    RBT4_STANDARD_WELD_DATA : WORD ;
    RBT5_STANDARD_WELD_DATA : WORD ;
    RBT6_STANDARD_WELD_DATA : WORD ;
    RBT7_STANDARD_WELD_DATA : WORD ;
    RBT8_STANDARD_WELD_DATA : WORD ;
    RBT9_STANDARD_WELD_DATA : WORD ;
    RBT10_STANDARD_WELD_DATA : WORD ;
    RBT11_STANDARD_WELD_DATA : WORD ;
    RBT12_STANDARD_WELD_DATA : WORD ;
    RBT13_STANDARD_WELD_DATA : WORD ;
    RBT14_STANDARD_WELD_DATA : WORD ;
    RBT15_STANDARD_WELD_DATA : WORD ;
    RBT16_STANDARD_WELD_DATA : WORD ;
    RBT17_STANDARD_WELD_DATA : WORD ;
    RBT18_STANDARD_WELD_DATA : WORD ;
    RBT19_STANDARD_WELD_DATA : WORD ;
    RBT20_STANDARD_WELD_DATA : WORD ;
    RBT21_STANDARD_WELD_DATA : WORD ;
    RBT22_STANDARD_WELD_DATA : WORD ;
    RBT23_STANDARD_WELD_DAT : WORD ;
    RBT24_STANDARD_WELD_DAT : WORD ;
    CHK_WORD : WORD ;
    TEST_TEMP : ARRAY  [1 .. 40 ] OF BYTE ;
   END_STRUCT ;
   S701_BT_CODE_2016 : STRUCT
    STATION_MAIN : WORD ;
    DISTINCTION_LH_RH : WORD ;
    STAION_NUMBER : WORD ;
    BODY_TYPE_1ST : WORD ;
    BODY_TYPE_OPTION : WORD ;
    RBT1_STANDARD_WELD_DATA : WORD ;
    RBT2_STANDARD_WELD_DATA : WORD ;
    RBT3_STANDARD_WELD_DATA : WORD ;
    RBT4_STANDARD_WELD_DATA : WORD ;
    RBT5_STANDARD_WELD_DATA : WORD ;
    RBT6_STANDARD_WELD_DATA : WORD ;
    RBT7_STANDARD_WELD_DATA : WORD ;
    RBT8_STANDARD_WELD_DATA : WORD ;
    RBT9_STANDARD_WELD_DATA : WORD ;
    RBT10_STANDARD_WELD_DATA : WORD ;
    RBT11_STANDARD_WELD_DATA : WORD ;
    RBT12_STANDARD_WELD_DATA : WORD ;
    RBT13_STANDARD_WELD_DATA : WORD ;
    RBT14_STANDARD_WELD_DATA : WORD ;
    RBT15_STANDARD_WELD_DATA : WORD ;
    RBT16_STANDARD_WELD_DATA : WORD ;
    RBT17_STANDARD_WELD_DATA : WORD ;
    RBT18_STANDARD_WELD_DATA : WORD ;
    RBT19_STANDARD_WELD_DATA : WORD ;
    RBT20_STANDARD_WELD_DATA : WORD ;
    RBT21_STANDARD_WELD_DATA : WORD ;
    RBT22_STANDARD_WELD_DATA : WORD ;
    RBT23_STANDARD_WELD_DAT : WORD ;
    RBT24_STANDARD_WELD_DAT : WORD ;
    CHK_WORD : WORD ;
    TEST_TEMP : ARRAY  [1 .. 40 ] OF BYTE ;
   END_STRUCT ;
   S701_BT_CODE_2017 : STRUCT
    STATION_MAIN : WORD ;
    DISTINCTION_LH_RH : WORD ;
    STAION_NUMBER : WORD ;
    BODY_TYPE_1ST : WORD ;
    BODY_TYPE_OPTION : WORD ;
    RBT1_STANDARD_WELD_DATA : WORD ;
    RBT2_STANDARD_WELD_DATA : WORD ;
    RBT3_STANDARD_WELD_DATA : WORD ;
    RBT4_STANDARD_WELD_DATA : WORD ;
    RBT5_STANDARD_WELD_DATA : WORD ;
    RBT6_STANDARD_WELD_DATA : WORD ;
    RBT7_STANDARD_WELD_DATA : WORD ;
    RBT8_STANDARD_WELD_DATA : WORD ;
    RBT9_STANDARD_WELD_DATA : WORD ;
    RBT10_STANDARD_WELD_DATA : WORD ;
    RBT11_STANDARD_WELD_DATA : WORD ;
    RBT12_STANDARD_WELD_DATA : WORD ;
    RBT13_STANDARD_WELD_DATA : WORD ;
    RBT14_STANDARD_WELD_DATA : WORD ;
    RBT15_STANDARD_WELD_DATA : WORD ;
    RBT16_STANDARD_WELD_DATA : WORD ;
    RBT17_STANDARD_WELD_DATA : WORD ;
    RBT18_STANDARD_WELD_DATA : WORD ;
    RBT19_STANDARD_WELD_DATA : WORD ;
    RBT20_STANDARD_WELD_DATA : WORD ;
    RBT21_STANDARD_WELD_DATA : WORD ;
    RBT22_STANDARD_WELD_DATA : WORD ;
    RBT23_STANDARD_WELD_DAT : WORD ;
    RBT24_STANDARD_WELD_DAT : WORD ;
    CHK_WORD : WORD ;
    TEST_TEMP : ARRAY  [1 .. 40 ] OF BYTE ;
   END_STRUCT ;
   S701_BT_CODE_2018 : STRUCT
    STATION_MAIN : WORD ;
    DISTINCTION_LH_RH : WORD ;
    STAION_NUMBER : WORD ;
    BODY_TYPE_1ST : WORD ;
    BODY_TYPE_OPTION : WORD ;
    RBT1_STANDARD_WELD_DATA : WORD ;
    RBT2_STANDARD_WELD_DATA : WORD ;
    RBT3_STANDARD_WELD_DATA : WORD ;
    RBT4_STANDARD_WELD_DATA : WORD ;
    RBT5_STANDARD_WELD_DATA : WORD ;
    RBT6_STANDARD_WELD_DATA : WORD ;
    RBT7_STANDARD_WELD_DATA : WORD ;
    RBT8_STANDARD_WELD_DATA : WORD ;
    RBT9_STANDARD_WELD_DATA : WORD ;
    RBT10_STANDARD_WELD_DATA : WORD ;
    RBT11_STANDARD_WELD_DATA : WORD ;
    RBT12_STANDARD_WELD_DATA : WORD ;
    RBT13_STANDARD_WELD_DATA : WORD ;
    RBT14_STANDARD_WELD_DATA : WORD ;
    RBT15_STANDARD_WELD_DATA : WORD ;
    RBT16_STANDARD_WELD_DATA : WORD ;
    RBT17_STANDARD_WELD_DATA : WORD ;
    RBT18_STANDARD_WELD_DATA : WORD ;
    RBT19_STANDARD_WELD_DATA : WORD ;
    RBT20_STANDARD_WELD_DATA : WORD ;
    RBT21_STANDARD_WELD_DATA : WORD ;
    RBT22_STANDARD_WELD_DATA : WORD ;
    RBT23_STANDARD_WELD_DAT : WORD ;
    RBT24_STANDARD_WELD_DAT : WORD ;
    CHK_WORD : WORD ;
    TEST_TEMP : ARRAY  [1 .. 40 ] OF BYTE ;
   END_STRUCT ;
   S701_BT_CODE_2019 : STRUCT
    STATION_MAIN : WORD ;
    DISTINCTION_LH_RH : WORD ;
    STAION_NUMBER : WORD ;
    BODY_TYPE_1ST : WORD ;
    BODY_TYPE_OPTION : WORD ;
    RBT1_STANDARD_WELD_DATA : WORD ;
    RBT2_STANDARD_WELD_DATA : WORD ;
    RBT3_STANDARD_WELD_DATA : WORD ;
    RBT4_STANDARD_WELD_DATA : WORD ;
    RBT5_STANDARD_WELD_DATA : WORD ;
    RBT6_STANDARD_WELD_DATA : WORD ;
    RBT7_STANDARD_WELD_DATA : WORD ;
    RBT8_STANDARD_WELD_DATA : WORD ;
    RBT9_STANDARD_WELD_DATA : WORD ;
    RBT10_STANDARD_WELD_DATA : WORD ;
    RBT11_STANDARD_WELD_DATA : WORD ;
    RBT12_STANDARD_WELD_DATA : WORD ;
    RBT13_STANDARD_WELD_DATA : WORD ;
    RBT14_STANDARD_WELD_DATA : WORD ;
    RBT15_STANDARD_WELD_DATA : WORD ;
    RBT16_STANDARD_WELD_DATA : WORD ;
    RBT17_STANDARD_WELD_DATA : WORD ;
    RBT18_STANDARD_WELD_DATA : WORD ;
    RBT19_STANDARD_WELD_DATA : WORD ;
    RBT20_STANDARD_WELD_DATA : WORD ;
    RBT21_STANDARD_WELD_DATA : WORD ;
    RBT22_STANDARD_WELD_DATA : WORD ;
    RBT23_STANDARD_WELD_DAT : WORD ;
    RBT24_STANDARD_WELD_DAT : WORD ;
    CHK_WORD : WORD ;
    TEST_TEMP : ARRAY  [1 .. 40 ] OF BYTE ;
   END_STRUCT ;
   S701_BT_CODE_2020 : STRUCT
    STATION_MAIN : WORD ;
    DISTINCTION_LH_RH : WORD ;
    STAION_NUMBER : WORD ;
    BODY_TYPE_1ST : WORD ;
    BODY_TYPE_OPTION : WORD ;
    RBT1_STANDARD_WELD_DATA : WORD ;
    RBT2_STANDARD_WELD_DATA : WORD ;
    RBT3_STANDARD_WELD_DATA : WORD ;
    RBT4_STANDARD_WELD_DATA : WORD ;
    RBT5_STANDARD_WELD_DATA : WORD ;
    RBT6_STANDARD_WELD_DATA : WORD ;
    RBT7_STANDARD_WELD_DATA : WORD ;
    RBT8_STANDARD_WELD_DATA : WORD ;
    RBT9_STANDARD_WELD_DATA : WORD ;
    RBT10_STANDARD_WELD_DATA : WORD ;
    RBT11_STANDARD_WELD_DATA : WORD ;
    RBT12_STANDARD_WELD_DATA : WORD ;
    RBT13_STANDARD_WELD_DATA : WORD ;
    RBT14_STANDARD_WELD_DATA : WORD ;
    RBT15_STANDARD_WELD_DATA : WORD ;
    RBT16_STANDARD_WELD_DATA : WORD ;
    RBT17_STANDARD_WELD_DATA : WORD ;
    RBT18_STANDARD_WELD_DATA : WORD ;
    RBT19_STANDARD_WELD_DATA : WORD ;
    RBT20_STANDARD_WELD_DATA : WORD ;
    RBT21_STANDARD_WELD_DATA : WORD ;
    RBT22_STANDARD_WELD_DATA : WORD ;
    RBT23_STANDARD_WELD_DAT : WORD ;
    RBT24_STANDARD_WELD_DAT : WORD ;
    CHK_WORD : WORD ;
    TEST_TEMP : ARRAY  [1 .. 40 ] OF BYTE ;
   END_STRUCT ;
   S701_BT_CODE_2021 : STRUCT
    STATION_MAIN : WORD ;
    DISTINCTION_LH_RH : WORD ;
    STAION_NUMBER : WORD ;
    BODY_TYPE_1ST : WORD ;
    BODY_TYPE_OPTION : WORD ;
    RBT1_STANDARD_WELD_DATA : WORD ;
    RBT2_STANDARD_WELD_DATA : WORD ;
    RBT3_STANDARD_WELD_DATA : WORD ;
    RBT4_STANDARD_WELD_DATA : WORD ;
    RBT5_STANDARD_WELD_DATA : WORD ;
    RBT6_STANDARD_WELD_DATA : WORD ;
    RBT7_STANDARD_WELD_DATA : WORD ;
    RBT8_STANDARD_WELD_DATA : WORD ;
    RBT9_STANDARD_WELD_DATA : WORD ;
    RBT10_STANDARD_WELD_DATA : WORD ;
    RBT11_STANDARD_WELD_DATA : WORD ;
    RBT12_STANDARD_WELD_DATA : WORD ;
    RBT13_STANDARD_WELD_DATA : WORD ;
    RBT14_STANDARD_WELD_DATA : WORD ;
    RBT15_STANDARD_WELD_DATA : WORD ;
    RBT16_STANDARD_WELD_DATA : WORD ;
    RBT17_STANDARD_WELD_DATA : WORD ;
    RBT18_STANDARD_WELD_DATA : WORD ;
    RBT19_STANDARD_WELD_DATA : WORD ;
    RBT20_STANDARD_WELD_DATA : WORD ;
    RBT21_STANDARD_WELD_DATA : WORD ;
    RBT22_STANDARD_WELD_DATA : WORD ;
    RBT23_STANDARD_WELD_DAT : WORD ;
    RBT24_STANDARD_WELD_DAT : WORD ;
    CHK_WORD : WORD ;
    TEST_TEMP : ARRAY  [1 .. 40 ] OF BYTE ;
   END_STRUCT ;
   S701_BT_CODE_2022 : STRUCT
    STATION_MAIN : WORD ;
    DISTINCTION_LH_RH : WORD ;
    STAION_NUMBER : WORD ;
    BODY_TYPE_1ST : WORD ;
    BODY_TYPE_OPTION : WORD ;
    RBT1_STANDARD_WELD_DATA : WORD ;
    RBT2_STANDARD_WELD_DATA : WORD ;
    RBT3_STANDARD_WELD_DATA : WORD ;
    RBT4_STANDARD_WELD_DATA : WORD ;
    RBT5_STANDARD_WELD_DATA : WORD ;
    RBT6_STANDARD_WELD_DATA : WORD ;
    RBT7_STANDARD_WELD_DATA : WORD ;
    RBT8_STANDARD_WELD_DATA : WORD ;
    RBT9_STANDARD_WELD_DATA : WORD ;
    RBT10_STANDARD_WELD_DATA : WORD ;
    RBT11_STANDARD_WELD_DATA : WORD ;
    RBT12_STANDARD_WELD_DATA : WORD ;
    RBT13_STANDARD_WELD_DATA : WORD ;
    RBT14_STANDARD_WELD_DATA : WORD ;
    RBT15_STANDARD_WELD_DATA : WORD ;
    RBT16_STANDARD_WELD_DATA : WORD ;
    RBT17_STANDARD_WELD_DATA : WORD ;
    RBT18_STANDARD_WELD_DATA : WORD ;
    RBT19_STANDARD_WELD_DATA : WORD ;
    RBT20_STANDARD_WELD_DATA : WORD ;
    RBT21_STANDARD_WELD_DATA : WORD ;
    RBT22_STANDARD_WELD_DATA : WORD ;
    RBT23_STANDARD_WELD_DAT : WORD ;
    RBT24_STANDARD_WELD_DAT : WORD ;
    CHK_WORD : WORD ;
    TEST_TEMP : ARRAY  [1 .. 40 ] OF BYTE ;
   END_STRUCT ;
   S701_BT_CODE_2023 : STRUCT
    STATION_MAIN : WORD ;
    DISTINCTION_LH_RH : WORD ;
    STAION_NUMBER : WORD ;
    BODY_TYPE_1ST : WORD ;
    BODY_TYPE_OPTION : WORD ;
    RBT1_STANDARD_WELD_DATA : WORD ;
    RBT2_STANDARD_WELD_DATA : WORD ;
    RBT3_STANDARD_WELD_DATA : WORD ;
    RBT4_STANDARD_WELD_DATA : WORD ;
    RBT5_STANDARD_WELD_DATA : WORD ;
    RBT6_STANDARD_WELD_DATA : WORD ;
    RBT7_STANDARD_WELD_DATA : WORD ;
    RBT8_STANDARD_WELD_DATA : WORD ;
    RBT9_STANDARD_WELD_DATA : WORD ;
    RBT10_STANDARD_WELD_DATA : WORD ;
    RBT11_STANDARD_WELD_DATA : WORD ;
    RBT12_STANDARD_WELD_DATA : WORD ;
    RBT13_STANDARD_WELD_DATA : WORD ;
    RBT14_STANDARD_WELD_DATA : WORD ;
    RBT15_STANDARD_WELD_DATA : WORD ;
    RBT16_STANDARD_WELD_DATA : WORD ;
    RBT17_STANDARD_WELD_DATA : WORD ;
    RBT18_STANDARD_WELD_DATA : WORD ;
    RBT19_STANDARD_WELD_DATA : WORD ;
    RBT20_STANDARD_WELD_DATA : WORD ;
    RBT21_STANDARD_WELD_DATA : WORD ;
    RBT22_STANDARD_WELD_DATA : WORD ;
    RBT23_STANDARD_WELD_DAT : WORD ;
    RBT24_STANDARD_WELD_DAT : WORD ;
    CHK_WORD : WORD ;
    TEST_TEMP : ARRAY  [1 .. 40 ] OF BYTE ;
   END_STRUCT ;
   S701_BT_CODE_2024 : STRUCT
    STATION_MAIN : WORD ;
    DISTINCTION_LH_RH : WORD ;
    STAION_NUMBER : WORD ;
    BODY_TYPE_1ST : WORD ;
    BODY_TYPE_OPTION : WORD ;
    RBT1_STANDARD_WELD_DATA : WORD ;
    RBT2_STANDARD_WELD_DATA : WORD ;
    RBT3_STANDARD_WELD_DATA : WORD ;
    RBT4_STANDARD_WELD_DATA : WORD ;
    RBT5_STANDARD_WELD_DATA : WORD ;
    RBT6_STANDARD_WELD_DATA : WORD ;
    RBT7_STANDARD_WELD_DATA : WORD ;
    RBT8_STANDARD_WELD_DATA : WORD ;
    RBT9_STANDARD_WELD_DATA : WORD ;
    RBT10_STANDARD_WELD_DATA : WORD ;
    RBT11_STANDARD_WELD_DATA : WORD ;
    RBT12_STANDARD_WELD_DATA : WORD ;
    RBT13_STANDARD_WELD_DATA : WORD ;
    RBT14_STANDARD_WELD_DATA : WORD ;
    RBT15_STANDARD_WELD_DATA : WORD ;
    RBT16_STANDARD_WELD_DATA : WORD ;
    RBT17_STANDARD_WELD_DATA : WORD ;
    RBT18_STANDARD_WELD_DATA : WORD ;
    RBT19_STANDARD_WELD_DATA : WORD ;
    RBT20_STANDARD_WELD_DATA : WORD ;
    RBT21_STANDARD_WELD_DATA : WORD ;
    RBT22_STANDARD_WELD_DATA : WORD ;
    RBT23_STANDARD_WELD_DAT : WORD ;
    RBT24_STANDARD_WELD_DAT : WORD ;
    CHK_WORD : WORD ;
    TEST_TEMP : ARRAY  [1 .. 40 ] OF BYTE ;
   END_STRUCT ;
   S701_BT_CODE_2025 : STRUCT
    STATION_MAIN : WORD ;
    DISTINCTION_LH_RH : WORD ;
    STAION_NUMBER : WORD ;
    BODY_TYPE_1ST : WORD ;
    BODY_TYPE_OPTION : WORD ;
    RBT1_STANDARD_WELD_DATA : WORD ;
    RBT2_STANDARD_WELD_DATA : WORD ;
    RBT3_STANDARD_WELD_DATA : WORD ;
    RBT4_STANDARD_WELD_DATA : WORD ;
    RBT5_STANDARD_WELD_DATA : WORD ;
    RBT6_STANDARD_WELD_DATA : WORD ;
    RBT7_STANDARD_WELD_DATA : WORD ;
    RBT8_STANDARD_WELD_DATA : WORD ;
    RBT9_STANDARD_WELD_DATA : WORD ;
    RBT10_STANDARD_WELD_DATA : WORD ;
    RBT11_STANDARD_WELD_DATA : WORD ;
    RBT12_STANDARD_WELD_DATA : WORD ;
    RBT13_STANDARD_WELD_DATA : WORD ;
    RBT14_STANDARD_WELD_DATA : WORD ;
    RBT15_STANDARD_WELD_DATA : WORD ;
    RBT16_STANDARD_WELD_DATA : WORD ;
    RBT17_STANDARD_WELD_DATA : WORD ;
    RBT18_STANDARD_WELD_DATA : WORD ;
    RBT19_STANDARD_WELD_DATA : WORD ;
    RBT20_STANDARD_WELD_DATA : WORD ;
    RBT21_STANDARD_WELD_DATA : WORD ;
    RBT22_STANDARD_WELD_DATA : WORD ;
    RBT23_STANDARD_WELD_DAT : WORD ;
    RBT24_STANDARD_WELD_DAT : WORD ;
    CHK_WORD : WORD ;
    TEST_TEMP : ARRAY  [1 .. 40 ] OF BYTE ;
   END_STRUCT ;
   S701_BT_CODE_2026 : STRUCT
    STATION_MAIN : WORD ;
    DISTINCTION_LH_RH : WORD ;
    STAION_NUMBER : WORD ;
    BODY_TYPE_1ST : WORD ;
    BODY_TYPE_OPTION : WORD ;
    RBT1_STANDARD_WELD_DATA : WORD ;
    RBT2_STANDARD_WELD_DATA : WORD ;
    RBT3_STANDARD_WELD_DATA : WORD ;
    RBT4_STANDARD_WELD_DATA : WORD ;
    RBT5_STANDARD_WELD_DATA : WORD ;
    RBT6_STANDARD_WELD_DATA : WORD ;
    RBT7_STANDARD_WELD_DATA : WORD ;
    RBT8_STANDARD_WELD_DATA : WORD ;
    RBT9_STANDARD_WELD_DATA : WORD ;
    RBT10_STANDARD_WELD_DATA : WORD ;
    RBT11_STANDARD_WELD_DATA : WORD ;
    RBT12_STANDARD_WELD_DATA : WORD ;
    RBT13_STANDARD_WELD_DATA : WORD ;
    RBT14_STANDARD_WELD_DATA : WORD ;
    RBT15_STANDARD_WELD_DATA : WORD ;
    RBT16_STANDARD_WELD_DATA : WORD ;
    RBT17_STANDARD_WELD_DATA : WORD ;
    RBT18_STANDARD_WELD_DATA : WORD ;
    RBT19_STANDARD_WELD_DATA : WORD ;
    RBT20_STANDARD_WELD_DATA : WORD ;
    RBT21_STANDARD_WELD_DATA : WORD ;
    RBT22_STANDARD_WELD_DATA : WORD ;
    RBT23_STANDARD_WELD_DAT : WORD ;
    RBT24_STANDARD_WELD_DAT : WORD ;
    CHK_WORD : WORD ;
    TEST_TEMP : ARRAY  [1 .. 40 ] OF BYTE ;
   END_STRUCT ;
   S701_BT_CODE_2027 : STRUCT
    STATION_MAIN : WORD ;
    DISTINCTION_LH_RH : WORD ;
    STAION_NUMBER : WORD ;
    BODY_TYPE_1ST : WORD ;
    BODY_TYPE_OPTION : WORD ;
    RBT1_STANDARD_WELD_DATA : WORD ;
    RBT2_STANDARD_WELD_DATA : WORD ;
    RBT3_STANDARD_WELD_DATA : WORD ;
    RBT4_STANDARD_WELD_DATA : WORD ;
    RBT5_STANDARD_WELD_DATA : WORD ;
    RBT6_STANDARD_WELD_DATA : WORD ;
    RBT7_STANDARD_WELD_DATA : WORD ;
    RBT8_STANDARD_WELD_DATA : WORD ;
    RBT9_STANDARD_WELD_DATA : WORD ;
    RBT10_STANDARD_WELD_DATA : WORD ;
    RBT11_STANDARD_WELD_DATA : WORD ;
    RBT12_STANDARD_WELD_DATA : WORD ;
    RBT13_STANDARD_WELD_DATA : WORD ;
    RBT14_STANDARD_WELD_DATA : WORD ;
    RBT15_STANDARD_WELD_DATA : WORD ;
    RBT16_STANDARD_WELD_DATA : WORD ;
    RBT17_STANDARD_WELD_DATA : WORD ;
    RBT18_STANDARD_WELD_DATA : WORD ;
    RBT19_STANDARD_WELD_DATA : WORD ;
    RBT20_STANDARD_WELD_DATA : WORD ;
    RBT21_STANDARD_WELD_DATA : WORD ;
    RBT22_STANDARD_WELD_DATA : WORD ;
    RBT23_STANDARD_WELD_DAT : WORD ;
    RBT24_STANDARD_WELD_DAT : WORD ;
    CHK_WORD : WORD ;
    TEST_TEMP : ARRAY  [1 .. 40 ] OF BYTE ;
   END_STRUCT ;
   S701_BT_CODE_2028 : STRUCT
    STATION_MAIN : WORD ;
    DISTINCTION_LH_RH : WORD ;
    STAION_NUMBER : WORD ;
    BODY_TYPE_1ST : WORD ;
    BODY_TYPE_OPTION : WORD ;
    RBT1_STANDARD_WELD_DATA : WORD ;
    RBT2_STANDARD_WELD_DATA : WORD ;
    RBT3_STANDARD_WELD_DATA : WORD ;
    RBT4_STANDARD_WELD_DATA : WORD ;
    RBT5_STANDARD_WELD_DATA : WORD ;
    RBT6_STANDARD_WELD_DATA : WORD ;
    RBT7_STANDARD_WELD_DATA : WORD ;
    RBT8_STANDARD_WELD_DATA : WORD ;
    RBT9_STANDARD_WELD_DATA : WORD ;
    RBT10_STANDARD_WELD_DATA : WORD ;
    RBT11_STANDARD_WELD_DATA : WORD ;
    RBT12_STANDARD_WELD_DATA : WORD ;
    RBT13_STANDARD_WELD_DATA : WORD ;
    RBT14_STANDARD_WELD_DATA : WORD ;
    RBT15_STANDARD_WELD_DATA : WORD ;
    RBT16_STANDARD_WELD_DATA : WORD ;
    RBT17_STANDARD_WELD_DATA : WORD ;
    RBT18_STANDARD_WELD_DATA : WORD ;
    RBT19_STANDARD_WELD_DATA : WORD ;
    RBT20_STANDARD_WELD_DATA : WORD ;
    RBT21_STANDARD_WELD_DATA : WORD ;
    RBT22_STANDARD_WELD_DATA : WORD ;
    RBT23_STANDARD_WELD_DAT : WORD ;
    RBT24_STANDARD_WELD_DAT : WORD ;
    CHK_WORD : WORD ;
    TEST_TEMP : ARRAY  [1 .. 40 ] OF BYTE ;
   END_STRUCT ;
   S701_BT_CODE_2029 : STRUCT
    STATION_MAIN : WORD ;
    DISTINCTION_LH_RH : WORD ;
    STAION_NUMBER : WORD ;
    BODY_TYPE_1ST : WORD ;
    BODY_TYPE_OPTION : WORD ;
    RBT1_STANDARD_WELD_DATA : WORD ;
    RBT2_STANDARD_WELD_DATA : WORD ;
    RBT3_STANDARD_WELD_DATA : WORD ;
    RBT4_STANDARD_WELD_DATA : WORD ;
    RBT5_STANDARD_WELD_DATA : WORD ;
    RBT6_STANDARD_WELD_DATA : WORD ;
    RBT7_STANDARD_WELD_DATA : WORD ;
    RBT8_STANDARD_WELD_DATA : WORD ;
    RBT9_STANDARD_WELD_DATA : WORD ;
    RBT10_STANDARD_WELD_DATA : WORD ;
    RBT11_STANDARD_WELD_DATA : WORD ;
    RBT12_STANDARD_WELD_DATA : WORD ;
    RBT13_STANDARD_WELD_DATA : WORD ;
    RBT14_STANDARD_WELD_DATA : WORD ;
    RBT15_STANDARD_WELD_DATA : WORD ;
    RBT16_STANDARD_WELD_DATA : WORD ;
    RBT17_STANDARD_WELD_DATA : WORD ;
    RBT18_STANDARD_WELD_DATA : WORD ;
    RBT19_STANDARD_WELD_DATA : WORD ;
    RBT20_STANDARD_WELD_DATA : WORD ;
    RBT21_STANDARD_WELD_DATA : WORD ;
    RBT22_STANDARD_WELD_DATA : WORD ;
    RBT23_STANDARD_WELD_DAT : WORD ;
    RBT24_STANDARD_WELD_DAT : WORD ;
    CHK_WORD : WORD ;
    TEST_TEMP : ARRAY  [1 .. 40 ] OF BYTE ;
   END_STRUCT ;
   S701_BT_CODE_2030 : STRUCT
    STATION_MAIN : WORD ;
    DISTINCTION_LH_RH : WORD ;
    STAION_NUMBER : WORD ;
    BODY_TYPE_1ST : WORD ;
    BODY_TYPE_OPTION : WORD ;
    RBT1_STANDARD_WELD_DATA : WORD ;
    RBT2_STANDARD_WELD_DATA : WORD ;
    RBT3_STANDARD_WELD_DATA : WORD ;
    RBT4_STANDARD_WELD_DATA : WORD ;
    RBT5_STANDARD_WELD_DATA : WORD ;
    RBT6_STANDARD_WELD_DATA : WORD ;
    RBT7_STANDARD_WELD_DATA : WORD ;
    RBT8_STANDARD_WELD_DATA : WORD ;
    RBT9_STANDARD_WELD_DATA : WORD ;
    RBT10_STANDARD_WELD_DATA : WORD ;
    RBT11_STANDARD_WELD_DATA : WORD ;
    RBT12_STANDARD_WELD_DATA : WORD ;
    RBT13_STANDARD_WELD_DATA : WORD ;
    RBT14_STANDARD_WELD_DATA : WORD ;
    RBT15_STANDARD_WELD_DATA : WORD ;
    RBT16_STANDARD_WELD_DATA : WORD ;
    RBT17_STANDARD_WELD_DATA : WORD ;
    RBT18_STANDARD_WELD_DATA : WORD ;
    RBT19_STANDARD_WELD_DATA : WORD ;
    RBT20_STANDARD_WELD_DATA : WORD ;
    RBT21_STANDARD_WELD_DATA : WORD ;
    RBT22_STANDARD_WELD_DATA : WORD ;
    RBT23_STANDARD_WELD_DAT : WORD ;
    RBT24_STANDARD_WELD_DAT : WORD ;
    CHK_WORD : WORD ;
    TEST_TEMP : ARRAY  [1 .. 40 ] OF BYTE ;
   END_STRUCT ;
   S700_BT_CODE_2101 : STRUCT
    STATION_MAIN : WORD ;
    DISTINCTION_LH_RH : WORD ;
    STAION_NUMBER : WORD ;
    BODY_TYPE_1ST : WORD ;
    BODY_TYPE_OPTION : WORD ;
    RBT1_STANDARD_WELD_DATA : WORD ;
    RBT2_STANDARD_WELD_DATA : WORD ;
    RBT3_STANDARD_WELD_DATA : WORD ;
    RBT4_STANDARD_WELD_DATA : WORD ;
    RBT5_STANDARD_WELD_DATA : WORD ;
    RBT6_STANDARD_WELD_DATA : WORD ;
    RBT7_STANDARD_WELD_DATA : WORD ;
    RBT8_STANDARD_WELD_DATA : WORD ;
    RBT9_STANDARD_WELD_DATA : WORD ;
    RBT10_STANDARD_WELD_DATA : WORD ;
    RBT11_STANDARD_WELD_DATA : WORD ;
    RBT12_STANDARD_WELD_DATA : WORD ;
    RBT13_STANDARD_WELD_DATA : WORD ;
    RBT14_STANDARD_WELD_DATA : WORD ;
    RBT15_STANDARD_WELD_DATA : WORD ;
    RBT16_STANDARD_WELD_DATA : WORD ;
    RBT17_STANDARD_WELD_DATA : WORD ;
    RBT18_STANDARD_WELD_DATA : WORD ;
    RBT19_STANDARD_WELD_DATA : WORD ;
    RBT20_STANDARD_WELD_DATA : WORD ;
    RBT21_STANDARD_WELD_DATA : WORD ;
    RBT22_STANDARD_WELD_DATA : WORD ;
    RBT23_STANDARD_WELD_DAT : WORD ;
    RBT24_STANDARD_WELD_DAT : WORD ;
    CHK_WORD : WORD ;
    TEST_TEMP : ARRAY  [1 .. 40 ] OF BYTE ;
   END_STRUCT ;
   S700_BT_CODE_2102 : STRUCT
    STATION_MAIN : WORD ;
    DISTINCTION_LH_RH : WORD ;
    STAION_NUMBER : WORD ;
    BODY_TYPE_1ST : WORD ;
    BODY_TYPE_OPTION : WORD ;
    RBT1_STANDARD_WELD_DATA : WORD ;
    RBT2_STANDARD_WELD_DATA : WORD ;
    RBT3_STANDARD_WELD_DATA : WORD ;
    RBT4_STANDARD_WELD_DATA : WORD ;
    RBT5_STANDARD_WELD_DATA : WORD ;
    RBT6_STANDARD_WELD_DATA : WORD ;
    RBT7_STANDARD_WELD_DATA : WORD ;
    RBT8_STANDARD_WELD_DATA : WORD ;
    RBT9_STANDARD_WELD_DATA : WORD ;
    RBT10_STANDARD_WELD_DATA : WORD ;
    RBT11_STANDARD_WELD_DATA : WORD ;
    RBT12_STANDARD_WELD_DATA : WORD ;
    RBT13_STANDARD_WELD_DATA : WORD ;
    RBT14_STANDARD_WELD_DATA : WORD ;
    RBT15_STANDARD_WELD_DATA : WORD ;
    RBT16_STANDARD_WELD_DATA : WORD ;
    RBT17_STANDARD_WELD_DATA : WORD ;
    RBT18_STANDARD_WELD_DATA : WORD ;
    RBT19_STANDARD_WELD_DATA : WORD ;
    RBT20_STANDARD_WELD_DATA : WORD ;
    RBT21_STANDARD_WELD_DATA : WORD ;
    RBT22_STANDARD_WELD_DATA : WORD ;
    RBT23_STANDARD_WELD_DAT : WORD ;
    RBT24_STANDARD_WELD_DAT : WORD ;
    CHK_WORD : WORD ;
    TEST_TEMP : ARRAY  [1 .. 40 ] OF BYTE ;
   END_STRUCT ;
   S700_BT_CODE_2103 : STRUCT
    STATION_MAIN : WORD ;
    DISTINCTION_LH_RH : WORD ;
    STAION_NUMBER : WORD ;
    BODY_TYPE_1ST : WORD ;
    BODY_TYPE_OPTION : WORD ;
    RBT1_STANDARD_WELD_DATA : WORD ;
    RBT2_STANDARD_WELD_DATA : WORD ;
    RBT3_STANDARD_WELD_DATA : WORD ;
    RBT4_STANDARD_WELD_DATA : WORD ;
    RBT5_STANDARD_WELD_DATA : WORD ;
    RBT6_STANDARD_WELD_DATA : WORD ;
    RBT7_STANDARD_WELD_DATA : WORD ;
    RBT8_STANDARD_WELD_DATA : WORD ;
    RBT9_STANDARD_WELD_DATA : WORD ;
    RBT10_STANDARD_WELD_DATA : WORD ;
    RBT11_STANDARD_WELD_DATA : WORD ;
    RBT12_STANDARD_WELD_DATA : WORD ;
    RBT13_STANDARD_WELD_DATA : WORD ;
    RBT14_STANDARD_WELD_DATA : WORD ;
    RBT15_STANDARD_WELD_DATA : WORD ;
    RBT16_STANDARD_WELD_DATA : WORD ;
    RBT17_STANDARD_WELD_DATA : WORD ;
    RBT18_STANDARD_WELD_DATA : WORD ;
    RBT19_STANDARD_WELD_DATA : WORD ;
    RBT20_STANDARD_WELD_DATA : WORD ;
    RBT21_STANDARD_WELD_DATA : WORD ;
    RBT22_STANDARD_WELD_DATA : WORD ;
    RBT23_STANDARD_WELD_DAT : WORD ;
    RBT24_STANDARD_WELD_DAT : WORD ;
    CHK_WORD : WORD ;
    TEST_TEMP : ARRAY  [1 .. 40 ] OF BYTE ;
   END_STRUCT ;
   S700_BT_CODE_2104 : STRUCT
    STATION_MAIN : WORD ;
    DISTINCTION_LH_RH : WORD ;
    STAION_NUMBER : WORD ;
    BODY_TYPE_1ST : WORD ;
    BODY_TYPE_OPTION : WORD ;
    RBT1_STANDARD_WELD_DATA : WORD ;
    RBT2_STANDARD_WELD_DATA : WORD ;
    RBT3_STANDARD_WELD_DATA : WORD ;
    RBT4_STANDARD_WELD_DATA : WORD ;
    RBT5_STANDARD_WELD_DATA : WORD ;
    RBT6_STANDARD_WELD_DATA : WORD ;
    RBT7_STANDARD_WELD_DATA : WORD ;
    RBT8_STANDARD_WELD_DATA : WORD ;
    RBT9_STANDARD_WELD_DATA : WORD ;
    RBT10_STANDARD_WELD_DATA : WORD ;
    RBT11_STANDARD_WELD_DATA : WORD ;
    RBT12_STANDARD_WELD_DATA : WORD ;
    RBT13_STANDARD_WELD_DATA : WORD ;
    RBT14_STANDARD_WELD_DATA : WORD ;
    RBT15_STANDARD_WELD_DATA : WORD ;
    RBT16_STANDARD_WELD_DATA : WORD ;
    RBT17_STANDARD_WELD_DATA : WORD ;
    RBT18_STANDARD_WELD_DATA : WORD ;
    RBT19_STANDARD_WELD_DATA : WORD ;
    RBT20_STANDARD_WELD_DATA : WORD ;
    RBT21_STANDARD_WELD_DATA : WORD ;
    RBT22_STANDARD_WELD_DATA : WORD ;
    RBT23_STANDARD_WELD_DAT : WORD ;
    RBT24_STANDARD_WELD_DAT : WORD ;
    CHK_WORD : WORD ;
    TEST_TEMP : ARRAY  [1 .. 40 ] OF BYTE ;
   END_STRUCT ;
   S700_BT_CODE_2105 : STRUCT
    STATION_MAIN : WORD ;
    DISTINCTION_LH_RH : WORD ;
    STAION_NUMBER : WORD ;
    BODY_TYPE_1ST : WORD ;
    BODY_TYPE_OPTION : WORD ;
    RBT1_STANDARD_WELD_DATA : WORD ;
    RBT2_STANDARD_WELD_DATA : WORD ;
    RBT3_STANDARD_WELD_DATA : WORD ;
    RBT4_STANDARD_WELD_DATA : WORD ;
    RBT5_STANDARD_WELD_DATA : WORD ;
    RBT6_STANDARD_WELD_DATA : WORD ;
    RBT7_STANDARD_WELD_DATA : WORD ;
    RBT8_STANDARD_WELD_DATA : WORD ;
    RBT9_STANDARD_WELD_DATA : WORD ;
    RBT10_STANDARD_WELD_DATA : WORD ;
    RBT11_STANDARD_WELD_DATA : WORD ;
    RBT12_STANDARD_WELD_DATA : WORD ;
    RBT13_STANDARD_WELD_DATA : WORD ;
    RBT14_STANDARD_WELD_DATA : WORD ;
    RBT15_STANDARD_WELD_DATA : WORD ;
    RBT16_STANDARD_WELD_DATA : WORD ;
    RBT17_STANDARD_WELD_DATA : WORD ;
    RBT18_STANDARD_WELD_DATA : WORD ;
    RBT19_STANDARD_WELD_DATA : WORD ;
    RBT20_STANDARD_WELD_DATA : WORD ;
    RBT21_STANDARD_WELD_DATA : WORD ;
    RBT22_STANDARD_WELD_DATA : WORD ;
    RBT23_STANDARD_WELD_DAT : WORD ;
    RBT24_STANDARD_WELD_DAT : WORD ;
    CHK_WORD : WORD ;
    TEST_TEMP : ARRAY  [1 .. 40 ] OF BYTE ;
   END_STRUCT ;
   S700_BT_CODE_2106 : STRUCT
    STATION_MAIN : WORD ;
    DISTINCTION_LH_RH : WORD ;
    STAION_NUMBER : WORD ;
    BODY_TYPE_1ST : WORD ;
    BODY_TYPE_OPTION : WORD ;
    RBT1_STANDARD_WELD_DATA : WORD ;
    RBT2_STANDARD_WELD_DATA : WORD ;
    RBT3_STANDARD_WELD_DATA : WORD ;
    RBT4_STANDARD_WELD_DATA : WORD ;
    RBT5_STANDARD_WELD_DATA : WORD ;
    RBT6_STANDARD_WELD_DATA : WORD ;
    RBT7_STANDARD_WELD_DATA : WORD ;
    RBT8_STANDARD_WELD_DATA : WORD ;
    RBT9_STANDARD_WELD_DATA : WORD ;
    RBT10_STANDARD_WELD_DATA : WORD ;
    RBT11_STANDARD_WELD_DATA : WORD ;
    RBT12_STANDARD_WELD_DATA : WORD ;
    RBT13_STANDARD_WELD_DATA : WORD ;
    RBT14_STANDARD_WELD_DATA : WORD ;
    RBT15_STANDARD_WELD_DATA : WORD ;
    RBT16_STANDARD_WELD_DATA : WORD ;
    RBT17_STANDARD_WELD_DATA : WORD ;
    RBT18_STANDARD_WELD_DATA : WORD ;
    RBT19_STANDARD_WELD_DATA : WORD ;
    RBT20_STANDARD_WELD_DATA : WORD ;
    RBT21_STANDARD_WELD_DATA : WORD ;
    RBT22_STANDARD_WELD_DATA : WORD ;
    RBT23_STANDARD_WELD_DAT : WORD ;
    RBT24_STANDARD_WELD_DAT : WORD ;
    CHK_WORD : WORD ;
    TEST_TEMP : ARRAY  [1 .. 40 ] OF BYTE ;
   END_STRUCT ;
   S700_BT_CODE_2107 : STRUCT
    STATION_MAIN : WORD ;
    DISTINCTION_LH_RH : WORD ;
    STAION_NUMBER : WORD ;
    BODY_TYPE_1ST : WORD ;
    BODY_TYPE_OPTION : WORD ;
    RBT1_STANDARD_WELD_DATA : WORD ;
    RBT2_STANDARD_WELD_DATA : WORD ;
    RBT3_STANDARD_WELD_DATA : WORD ;
    RBT4_STANDARD_WELD_DATA : WORD ;
    RBT5_STANDARD_WELD_DATA : WORD ;
    RBT6_STANDARD_WELD_DATA : WORD ;
    RBT7_STANDARD_WELD_DATA : WORD ;
    RBT8_STANDARD_WELD_DATA : WORD ;
    RBT9_STANDARD_WELD_DATA : WORD ;
    RBT10_STANDARD_WELD_DATA : WORD ;
    RBT11_STANDARD_WELD_DATA : WORD ;
    RBT12_STANDARD_WELD_DATA : WORD ;
    RBT13_STANDARD_WELD_DATA : WORD ;
    RBT14_STANDARD_WELD_DATA : WORD ;
    RBT15_STANDARD_WELD_DATA : WORD ;
    RBT16_STANDARD_WELD_DATA : WORD ;
    RBT17_STANDARD_WELD_DATA : WORD ;
    RBT18_STANDARD_WELD_DATA : WORD ;
    RBT19_STANDARD_WELD_DATA : WORD ;
    RBT20_STANDARD_WELD_DATA : WORD ;
    RBT21_STANDARD_WELD_DATA : WORD ;
    RBT22_STANDARD_WELD_DATA : WORD ;
    RBT23_STANDARD_WELD_DAT : WORD ;
    RBT24_STANDARD_WELD_DAT : WORD ;
    CHK_WORD : WORD ;
    TEST_TEMP : ARRAY  [1 .. 40 ] OF BYTE ;
   END_STRUCT ;
   S700_BT_CODE_2108 : STRUCT
    STATION_MAIN : WORD ;
    DISTINCTION_LH_RH : WORD ;
    STAION_NUMBER : WORD ;
    BODY_TYPE_1ST : WORD ;
    BODY_TYPE_OPTION : WORD ;
    RBT1_STANDARD_WELD_DATA : WORD ;
    RBT2_STANDARD_WELD_DATA : WORD ;
    RBT3_STANDARD_WELD_DATA : WORD ;
    RBT4_STANDARD_WELD_DATA : WORD ;
    RBT5_STANDARD_WELD_DATA : WORD ;
    RBT6_STANDARD_WELD_DATA : WORD ;
    RBT7_STANDARD_WELD_DATA : WORD ;
    RBT8_STANDARD_WELD_DATA : WORD ;
    RBT9_STANDARD_WELD_DATA : WORD ;
    RBT10_STANDARD_WELD_DATA : WORD ;
    RBT11_STANDARD_WELD_DATA : WORD ;
    RBT12_STANDARD_WELD_DATA : WORD ;
    RBT13_STANDARD_WELD_DATA : WORD ;
    RBT14_STANDARD_WELD_DATA : WORD ;
    RBT15_STANDARD_WELD_DATA : WORD ;
    RBT16_STANDARD_WELD_DATA : WORD ;
    RBT17_STANDARD_WELD_DATA : WORD ;
    RBT18_STANDARD_WELD_DATA : WORD ;
    RBT19_STANDARD_WELD_DATA : WORD ;
    RBT20_STANDARD_WELD_DATA : WORD ;
    RBT21_STANDARD_WELD_DATA : WORD ;
    RBT22_STANDARD_WELD_DATA : WORD ;
    RBT23_STANDARD_WELD_DAT : WORD ;
    RBT24_STANDARD_WELD_DAT : WORD ;
    CHK_WORD : WORD ;
    TEST_TEMP : ARRAY  [1 .. 40 ] OF BYTE ;
   END_STRUCT ;
   S700_BT_CODE_2109 : STRUCT
    STATION_MAIN : WORD ;
    DISTINCTION_LH_RH : WORD ;
    STAION_NUMBER : WORD ;
    BODY_TYPE_1ST : WORD ;
    BODY_TYPE_OPTION : WORD ;
    RBT1_STANDARD_WELD_DATA : WORD ;
    RBT2_STANDARD_WELD_DATA : WORD ;
    RBT3_STANDARD_WELD_DATA : WORD ;
    RBT4_STANDARD_WELD_DATA : WORD ;
    RBT5_STANDARD_WELD_DATA : WORD ;
    RBT6_STANDARD_WELD_DATA : WORD ;
    RBT7_STANDARD_WELD_DATA : WORD ;
    RBT8_STANDARD_WELD_DATA : WORD ;
    RBT9_STANDARD_WELD_DATA : WORD ;
    RBT10_STANDARD_WELD_DATA : WORD ;
    RBT11_STANDARD_WELD_DATA : WORD ;
    RBT12_STANDARD_WELD_DATA : WORD ;
    RBT13_STANDARD_WELD_DATA : WORD ;
    RBT14_STANDARD_WELD_DATA : WORD ;
    RBT15_STANDARD_WELD_DATA : WORD ;
    RBT16_STANDARD_WELD_DATA : WORD ;
    RBT17_STANDARD_WELD_DATA : WORD ;
    RBT18_STANDARD_WELD_DATA : WORD ;
    RBT19_STANDARD_WELD_DATA : WORD ;
    RBT20_STANDARD_WELD_DATA : WORD ;
    RBT21_STANDARD_WELD_DATA : WORD ;
    RBT22_STANDARD_WELD_DATA : WORD ;
    RBT23_STANDARD_WELD_DAT : WORD ;
    RBT24_STANDARD_WELD_DAT : WORD ;
    CHK_WORD : WORD ;
    TEST_TEMP : ARRAY  [1 .. 40 ] OF BYTE ;
   END_STRUCT ;
   S700_BT_CODE_2110 : STRUCT
    STATION_MAIN : WORD ;
    DISTINCTION_LH_RH : WORD ;
    STAION_NUMBER : WORD ;
    BODY_TYPE_1ST : WORD ;
    BODY_TYPE_OPTION : WORD ;
    RBT1_STANDARD_WELD_DATA : WORD ;
    RBT2_STANDARD_WELD_DATA : WORD ;
    RBT3_STANDARD_WELD_DATA : WORD ;
    RBT4_STANDARD_WELD_DATA : WORD ;
    RBT5_STANDARD_WELD_DATA : WORD ;
    RBT6_STANDARD_WELD_DATA : WORD ;
    RBT7_STANDARD_WELD_DATA : WORD ;
    RBT8_STANDARD_WELD_DATA : WORD ;
    RBT9_STANDARD_WELD_DATA : WORD ;
    RBT10_STANDARD_WELD_DATA : WORD ;
    RBT11_STANDARD_WELD_DATA : WORD ;
    RBT12_STANDARD_WELD_DATA : WORD ;
    RBT13_STANDARD_WELD_DATA : WORD ;
    RBT14_STANDARD_WELD_DATA : WORD ;
    RBT15_STANDARD_WELD_DATA : WORD ;
    RBT16_STANDARD_WELD_DATA : WORD ;
    RBT17_STANDARD_WELD_DATA : WORD ;
    RBT18_STANDARD_WELD_DATA : WORD ;
    RBT19_STANDARD_WELD_DATA : WORD ;
    RBT20_STANDARD_WELD_DATA : WORD ;
    RBT21_STANDARD_WELD_DATA : WORD ;
    RBT22_STANDARD_WELD_DATA : WORD ;
    RBT23_STANDARD_WELD_DAT : WORD ;
    RBT24_STANDARD_WELD_DAT : WORD ;
    CHK_WORD : WORD ;
    TEST_TEMP : ARRAY  [1 .. 40 ] OF BYTE ;
   END_STRUCT ;
   S700_BT_CODE_2111 : STRUCT
    STATION_MAIN : WORD ;
    DISTINCTION_LH_RH : WORD ;
    STAION_NUMBER : WORD ;
    BODY_TYPE_1ST : WORD ;
    BODY_TYPE_OPTION : WORD ;
    RBT1_STANDARD_WELD_DATA : WORD ;
    RBT2_STANDARD_WELD_DATA : WORD ;
    RBT3_STANDARD_WELD_DATA : WORD ;
    RBT4_STANDARD_WELD_DATA : WORD ;
    RBT5_STANDARD_WELD_DATA : WORD ;
    RBT6_STANDARD_WELD_DATA : WORD ;
    RBT7_STANDARD_WELD_DATA : WORD ;
    RBT8_STANDARD_WELD_DATA : WORD ;
    RBT9_STANDARD_WELD_DATA : WORD ;
    RBT10_STANDARD_WELD_DATA : WORD ;
    RBT11_STANDARD_WELD_DATA : WORD ;
    RBT12_STANDARD_WELD_DATA : WORD ;
    RBT13_STANDARD_WELD_DATA : WORD ;
    RBT14_STANDARD_WELD_DATA : WORD ;
    RBT15_STANDARD_WELD_DATA : WORD ;
    RBT16_STANDARD_WELD_DATA : WORD ;
    RBT17_STANDARD_WELD_DATA : WORD ;
    RBT18_STANDARD_WELD_DATA : WORD ;
    RBT19_STANDARD_WELD_DATA : WORD ;
    RBT20_STANDARD_WELD_DATA : WORD ;
    RBT21_STANDARD_WELD_DATA : WORD ;
    RBT22_STANDARD_WELD_DATA : WORD ;
    RBT23_STANDARD_WELD_DAT : WORD ;
    RBT24_STANDARD_WELD_DAT : WORD ;
    CHK_WORD : WORD ;
    TEST_TEMP : ARRAY  [1 .. 40 ] OF BYTE ;
   END_STRUCT ;
   S700_BT_CODE_2112 : STRUCT
    STATION_MAIN : WORD ;
    DISTINCTION_LH_RH : WORD ;
    STAION_NUMBER : WORD ;
    BODY_TYPE_1ST : WORD ;
    BODY_TYPE_OPTION : WORD ;
    RBT1_STANDARD_WELD_DATA : WORD ;
    RBT2_STANDARD_WELD_DATA : WORD ;
    RBT3_STANDARD_WELD_DATA : WORD ;
    RBT4_STANDARD_WELD_DATA : WORD ;
    RBT5_STANDARD_WELD_DATA : WORD ;
    RBT6_STANDARD_WELD_DATA : WORD ;
    RBT7_STANDARD_WELD_DATA : WORD ;
    RBT8_STANDARD_WELD_DATA : WORD ;
    RBT9_STANDARD_WELD_DATA : WORD ;
    RBT10_STANDARD_WELD_DATA : WORD ;
    RBT11_STANDARD_WELD_DATA : WORD ;
    RBT12_STANDARD_WELD_DATA : WORD ;
    RBT13_STANDARD_WELD_DATA : WORD ;
    RBT14_STANDARD_WELD_DATA : WORD ;
    RBT15_STANDARD_WELD_DATA : WORD ;
    RBT16_STANDARD_WELD_DATA : WORD ;
    RBT17_STANDARD_WELD_DATA : WORD ;
    RBT18_STANDARD_WELD_DATA : WORD ;
    RBT19_STANDARD_WELD_DATA : WORD ;
    RBT20_STANDARD_WELD_DATA : WORD ;
    RBT21_STANDARD_WELD_DATA : WORD ;
    RBT22_STANDARD_WELD_DATA : WORD ;
    RBT23_STANDARD_WELD_DAT : WORD ;
    RBT24_STANDARD_WELD_DAT : WORD ;
    CHK_WORD : WORD ;
    TEST_TEMP : ARRAY  [1 .. 40 ] OF BYTE ;
   END_STRUCT ;
   S700_BT_CODE_2113 : STRUCT
    STATION_MAIN : WORD ;
    DISTINCTION_LH_RH : WORD ;
    STAION_NUMBER : WORD ;
    BODY_TYPE_1ST : WORD ;
    BODY_TYPE_OPTION : WORD ;
    RBT1_STANDARD_WELD_DATA : WORD ;
    RBT2_STANDARD_WELD_DATA : WORD ;
    RBT3_STANDARD_WELD_DATA : WORD ;
    RBT4_STANDARD_WELD_DATA : WORD ;
    RBT5_STANDARD_WELD_DATA : WORD ;
    RBT6_STANDARD_WELD_DATA : WORD ;
    RBT7_STANDARD_WELD_DATA : WORD ;
    RBT8_STANDARD_WELD_DATA : WORD ;
    RBT9_STANDARD_WELD_DATA : WORD ;
    RBT10_STANDARD_WELD_DATA : WORD ;
    RBT11_STANDARD_WELD_DATA : WORD ;
    RBT12_STANDARD_WELD_DATA : WORD ;
    RBT13_STANDARD_WELD_DATA : WORD ;
    RBT14_STANDARD_WELD_DATA : WORD ;
    RBT15_STANDARD_WELD_DATA : WORD ;
    RBT16_STANDARD_WELD_DATA : WORD ;
    RBT17_STANDARD_WELD_DATA : WORD ;
    RBT18_STANDARD_WELD_DATA : WORD ;
    RBT19_STANDARD_WELD_DATA : WORD ;
    RBT20_STANDARD_WELD_DATA : WORD ;
    RBT21_STANDARD_WELD_DATA : WORD ;
    RBT22_STANDARD_WELD_DATA : WORD ;
    RBT23_STANDARD_WELD_DAT : WORD ;
    RBT24_STANDARD_WELD_DAT : WORD ;
    CHK_WORD : WORD ;
    TEST_TEMP : ARRAY  [1 .. 40 ] OF BYTE ;
   END_STRUCT ;
   S700_BT_CODE_2114 : STRUCT
    STATION_MAIN : WORD ;
    DISTINCTION_LH_RH : WORD ;
    STAION_NUMBER : WORD ;
    BODY_TYPE_1ST : WORD ;
    BODY_TYPE_OPTION : WORD ;
    RBT1_STANDARD_WELD_DATA : WORD ;
    RBT2_STANDARD_WELD_DATA : WORD ;
    RBT3_STANDARD_WELD_DATA : WORD ;
    RBT4_STANDARD_WELD_DATA : WORD ;
    RBT5_STANDARD_WELD_DATA : WORD ;
    RBT6_STANDARD_WELD_DATA : WORD ;
    RBT7_STANDARD_WELD_DATA : WORD ;
    RBT8_STANDARD_WELD_DATA : WORD ;
    RBT9_STANDARD_WELD_DATA : WORD ;
    RBT10_STANDARD_WELD_DATA : WORD ;
    RBT11_STANDARD_WELD_DATA : WORD ;
    RBT12_STANDARD_WELD_DATA : WORD ;
    RBT13_STANDARD_WELD_DATA : WORD ;
    RBT14_STANDARD_WELD_DATA : WORD ;
    RBT15_STANDARD_WELD_DATA : WORD ;
    RBT16_STANDARD_WELD_DATA : WORD ;
    RBT17_STANDARD_WELD_DATA : WORD ;
    RBT18_STANDARD_WELD_DATA : WORD ;
    RBT19_STANDARD_WELD_DATA : WORD ;
    RBT20_STANDARD_WELD_DATA : WORD ;
    RBT21_STANDARD_WELD_DATA : WORD ;
    RBT22_STANDARD_WELD_DATA : WORD ;
    RBT23_STANDARD_WELD_DAT : WORD ;
    RBT24_STANDARD_WELD_DAT : WORD ;
    CHK_WORD : WORD ;
    TEST_TEMP : ARRAY  [1 .. 40 ] OF BYTE ;
   END_STRUCT ;
   S700_BT_CODE_2115 : STRUCT
    STATION_MAIN : WORD ;
    DISTINCTION_LH_RH : WORD ;
    STAION_NUMBER : WORD ;
    BODY_TYPE_1ST : WORD ;
    BODY_TYPE_OPTION : WORD ;
    RBT1_STANDARD_WELD_DATA : WORD ;
    RBT2_STANDARD_WELD_DATA : WORD ;
    RBT3_STANDARD_WELD_DATA : WORD ;
    RBT4_STANDARD_WELD_DATA : WORD ;
    RBT5_STANDARD_WELD_DATA : WORD ;
    RBT6_STANDARD_WELD_DATA : WORD ;
    RBT7_STANDARD_WELD_DATA : WORD ;
    RBT8_STANDARD_WELD_DATA : WORD ;
    RBT9_STANDARD_WELD_DATA : WORD ;
    RBT10_STANDARD_WELD_DATA : WORD ;
    RBT11_STANDARD_WELD_DATA : WORD ;
    RBT12_STANDARD_WELD_DATA : WORD ;
    RBT13_STANDARD_WELD_DATA : WORD ;
    RBT14_STANDARD_WELD_DATA : WORD ;
    RBT15_STANDARD_WELD_DATA : WORD ;
    RBT16_STANDARD_WELD_DATA : WORD ;
    RBT17_STANDARD_WELD_DATA : WORD ;
    RBT18_STANDARD_WELD_DATA : WORD ;
    RBT19_STANDARD_WELD_DATA : WORD ;
    RBT20_STANDARD_WELD_DATA : WORD ;
    RBT21_STANDARD_WELD_DATA : WORD ;
    RBT22_STANDARD_WELD_DATA : WORD ;
    RBT23_STANDARD_WELD_DAT : WORD ;
    RBT24_STANDARD_WELD_DAT : WORD ;
    CHK_WORD : WORD ;
    TEST_TEMP : ARRAY  [1 .. 40 ] OF BYTE ;
   END_STRUCT ;
   S700_BT_CODE_2116 : STRUCT
    STATION_MAIN : WORD ;
    DISTINCTION_LH_RH : WORD ;
    STAION_NUMBER : WORD ;
    BODY_TYPE_1ST : WORD ;
    BODY_TYPE_OPTION : WORD ;
    RBT1_STANDARD_WELD_DATA : WORD ;
    RBT2_STANDARD_WELD_DATA : WORD ;
    RBT3_STANDARD_WELD_DATA : WORD ;
    RBT4_STANDARD_WELD_DATA : WORD ;
    RBT5_STANDARD_WELD_DATA : WORD ;
    RBT6_STANDARD_WELD_DATA : WORD ;
    RBT7_STANDARD_WELD_DATA : WORD ;
    RBT8_STANDARD_WELD_DATA : WORD ;
    RBT9_STANDARD_WELD_DATA : WORD ;
    RBT10_STANDARD_WELD_DATA : WORD ;
    RBT11_STANDARD_WELD_DATA : WORD ;
    RBT12_STANDARD_WELD_DATA : WORD ;
    RBT13_STANDARD_WELD_DATA : WORD ;
    RBT14_STANDARD_WELD_DATA : WORD ;
    RBT15_STANDARD_WELD_DATA : WORD ;
    RBT16_STANDARD_WELD_DATA : WORD ;
    RBT17_STANDARD_WELD_DATA : WORD ;
    RBT18_STANDARD_WELD_DATA : WORD ;
    RBT19_STANDARD_WELD_DATA : WORD ;
    RBT20_STANDARD_WELD_DATA : WORD ;
    RBT21_STANDARD_WELD_DATA : WORD ;
    RBT22_STANDARD_WELD_DATA : WORD ;
    RBT23_STANDARD_WELD_DAT : WORD ;
    RBT24_STANDARD_WELD_DAT : WORD ;
    CHK_WORD : WORD ;
    TEST_TEMP : ARRAY  [1 .. 40 ] OF BYTE ;
   END_STRUCT ;
   S700_BT_CODE_2117 : STRUCT
    STATION_MAIN : WORD ;
    DISTINCTION_LH_RH : WORD ;
    STAION_NUMBER : WORD ;
    BODY_TYPE_1ST : WORD ;
    BODY_TYPE_OPTION : WORD ;
    RBT1_STANDARD_WELD_DATA : WORD ;
    RBT2_STANDARD_WELD_DATA : WORD ;
    RBT3_STANDARD_WELD_DATA : WORD ;
    RBT4_STANDARD_WELD_DATA : WORD ;
    RBT5_STANDARD_WELD_DATA : WORD ;
    RBT6_STANDARD_WELD_DATA : WORD ;
    RBT7_STANDARD_WELD_DATA : WORD ;
    RBT8_STANDARD_WELD_DATA : WORD ;
    RBT9_STANDARD_WELD_DATA : WORD ;
    RBT10_STANDARD_WELD_DATA : WORD ;
    RBT11_STANDARD_WELD_DATA : WORD ;
    RBT12_STANDARD_WELD_DATA : WORD ;
    RBT13_STANDARD_WELD_DATA : WORD ;
    RBT14_STANDARD_WELD_DATA : WORD ;
    RBT15_STANDARD_WELD_DATA : WORD ;
    RBT16_STANDARD_WELD_DATA : WORD ;
    RBT17_STANDARD_WELD_DATA : WORD ;
    RBT18_STANDARD_WELD_DATA : WORD ;
    RBT19_STANDARD_WELD_DATA : WORD ;
    RBT20_STANDARD_WELD_DATA : WORD ;
    RBT21_STANDARD_WELD_DATA : WORD ;
    RBT22_STANDARD_WELD_DATA : WORD ;
    RBT23_STANDARD_WELD_DAT : WORD ;
    RBT24_STANDARD_WELD_DAT : WORD ;
    CHK_WORD : WORD ;
    TEST_TEMP : ARRAY  [1 .. 40 ] OF BYTE ;
   END_STRUCT ;
   S700_BT_CODE_2118 : STRUCT
    STATION_MAIN : WORD ;
    DISTINCTION_LH_RH : WORD ;
    STAION_NUMBER : WORD ;
    BODY_TYPE_1ST : WORD ;
    BODY_TYPE_OPTION : WORD ;
    RBT1_STANDARD_WELD_DATA : WORD ;
    RBT2_STANDARD_WELD_DATA : WORD ;
    RBT3_STANDARD_WELD_DATA : WORD ;
    RBT4_STANDARD_WELD_DATA : WORD ;
    RBT5_STANDARD_WELD_DATA : WORD ;
    RBT6_STANDARD_WELD_DATA : WORD ;
    RBT7_STANDARD_WELD_DATA : WORD ;
    RBT8_STANDARD_WELD_DATA : WORD ;
    RBT9_STANDARD_WELD_DATA : WORD ;
    RBT10_STANDARD_WELD_DATA : WORD ;
    RBT11_STANDARD_WELD_DATA : WORD ;
    RBT12_STANDARD_WELD_DATA : WORD ;
    RBT13_STANDARD_WELD_DATA : WORD ;
    RBT14_STANDARD_WELD_DATA : WORD ;
    RBT15_STANDARD_WELD_DATA : WORD ;
    RBT16_STANDARD_WELD_DATA : WORD ;
    RBT17_STANDARD_WELD_DATA : WORD ;
    RBT18_STANDARD_WELD_DATA : WORD ;
    RBT19_STANDARD_WELD_DATA : WORD ;
    RBT20_STANDARD_WELD_DATA : WORD ;
    RBT21_STANDARD_WELD_DATA : WORD ;
    RBT22_STANDARD_WELD_DATA : WORD ;
    RBT23_STANDARD_WELD_DAT : WORD ;
    RBT24_STANDARD_WELD_DAT : WORD ;
    CHK_WORD : WORD ;
    TEST_TEMP : ARRAY  [1 .. 40 ] OF BYTE ;
   END_STRUCT ;
   S700_BT_CODE_2119 : STRUCT
    STATION_MAIN : WORD ;
    DISTINCTION_LH_RH : WORD ;
    STAION_NUMBER : WORD ;
    BODY_TYPE_1ST : WORD ;
    BODY_TYPE_OPTION : WORD ;
    RBT1_STANDARD_WELD_DATA : WORD ;
    RBT2_STANDARD_WELD_DATA : WORD ;
    RBT3_STANDARD_WELD_DATA : WORD ;
    RBT4_STANDARD_WELD_DATA : WORD ;
    RBT5_STANDARD_WELD_DATA : WORD ;
    RBT6_STANDARD_WELD_DATA : WORD ;
    RBT7_STANDARD_WELD_DATA : WORD ;
    RBT8_STANDARD_WELD_DATA : WORD ;
    RBT9_STANDARD_WELD_DATA : WORD ;
    RBT10_STANDARD_WELD_DATA : WORD ;
    RBT11_STANDARD_WELD_DATA : WORD ;
    RBT12_STANDARD_WELD_DATA : WORD ;
    RBT13_STANDARD_WELD_DATA : WORD ;
    RBT14_STANDARD_WELD_DATA : WORD ;
    RBT15_STANDARD_WELD_DATA : WORD ;
    RBT16_STANDARD_WELD_DATA : WORD ;
    RBT17_STANDARD_WELD_DATA : WORD ;
    RBT18_STANDARD_WELD_DATA : WORD ;
    RBT19_STANDARD_WELD_DATA : WORD ;
    RBT20_STANDARD_WELD_DATA : WORD ;
    RBT21_STANDARD_WELD_DATA : WORD ;
    RBT22_STANDARD_WELD_DATA : WORD ;
    RBT23_STANDARD_WELD_DAT : WORD ;
    RBT24_STANDARD_WELD_DAT : WORD ;
    CHK_WORD : WORD ;
    TEST_TEMP : ARRAY  [1 .. 40 ] OF BYTE ;
   END_STRUCT ;
   S700_BT_CODE_2120 : STRUCT
    STATION_MAIN : WORD ;
    DISTINCTION_LH_RH : WORD ;
    STAION_NUMBER : WORD ;
    BODY_TYPE_1ST : WORD ;
    BODY_TYPE_OPTION : WORD ;
    RBT1_STANDARD_WELD_DATA : WORD ;
    RBT2_STANDARD_WELD_DATA : WORD ;
    RBT3_STANDARD_WELD_DATA : WORD ;
    RBT4_STANDARD_WELD_DATA : WORD ;
    RBT5_STANDARD_WELD_DATA : WORD ;
    RBT6_STANDARD_WELD_DATA : WORD ;
    RBT7_STANDARD_WELD_DATA : WORD ;
    RBT8_STANDARD_WELD_DATA : WORD ;
    RBT9_STANDARD_WELD_DATA : WORD ;
    RBT10_STANDARD_WELD_DATA : WORD ;
    RBT11_STANDARD_WELD_DATA : WORD ;
    RBT12_STANDARD_WELD_DATA : WORD ;
    RBT13_STANDARD_WELD_DATA : WORD ;
    RBT14_STANDARD_WELD_DATA : WORD ;
    RBT15_STANDARD_WELD_DATA : WORD ;
    RBT16_STANDARD_WELD_DATA : WORD ;
    RBT17_STANDARD_WELD_DATA : WORD ;
    RBT18_STANDARD_WELD_DATA : WORD ;
    RBT19_STANDARD_WELD_DATA : WORD ;
    RBT20_STANDARD_WELD_DATA : WORD ;
    RBT21_STANDARD_WELD_DATA : WORD ;
    RBT22_STANDARD_WELD_DATA : WORD ;
    RBT23_STANDARD_WELD_DAT : WORD ;
    RBT24_STANDARD_WELD_DAT : WORD ;
    CHK_WORD : WORD ;
    TEST_TEMP : ARRAY  [1 .. 40 ] OF BYTE ;
   END_STRUCT ;
   S700_1_BT_CODE_2101 : STRUCT
    STATION_MAIN : WORD ;
    DISTINCTION_LH_RH : WORD ;
    STAION_NUMBER : WORD ;
    BODY_TYPE_1ST : WORD ;
    BODY_TYPE_OPTION : WORD ;
    RBT1_STANDARD_WELD_DATA : WORD ;
    RBT2_STANDARD_WELD_DATA : WORD ;
    RBT3_STANDARD_WELD_DATA : WORD ;
    RBT4_STANDARD_WELD_DATA : WORD ;
    RBT5_STANDARD_WELD_DATA : WORD ;
    RBT6_STANDARD_WELD_DATA : WORD ;
    RBT7_STANDARD_WELD_DATA : WORD ;
    RBT8_STANDARD_WELD_DATA : WORD ;
    RBT9_STANDARD_WELD_DATA : WORD ;
    RBT10_STANDARD_WELD_DATA : WORD ;
    RBT11_STANDARD_WELD_DATA : WORD ;
    RBT12_STANDARD_WELD_DATA : WORD ;
    RBT13_STANDARD_WELD_DATA : WORD ;
    RBT14_STANDARD_WELD_DATA : WORD ;
    RBT15_STANDARD_WELD_DATA : WORD ;
    RBT16_STANDARD_WELD_DATA : WORD ;
    RBT17_STANDARD_WELD_DATA : WORD ;
    RBT18_STANDARD_WELD_DATA : WORD ;
    RBT19_STANDARD_WELD_DATA : WORD ;
    RBT20_STANDARD_WELD_DATA : WORD ;
    RBT21_STANDARD_WELD_DATA : WORD ;
    RBT22_STANDARD_WELD_DATA : WORD ;
    RBT23_STANDARD_WELD_DAT : WORD ;
    RBT24_STANDARD_WELD_DAT : WORD ;
    CHK_WORD : WORD ;
    TEST_TEMP : ARRAY  [1 .. 40 ] OF BYTE ;
   END_STRUCT ;
   S700_1_BT_CODE_2102 : STRUCT
    STATION_MAIN : WORD ;
    DISTINCTION_LH_RH : WORD ;
    STAION_NUMBER : WORD ;
    BODY_TYPE_1ST : WORD ;
    BODY_TYPE_OPTION : WORD ;
    RBT1_STANDARD_WELD_DATA : WORD ;
    RBT2_STANDARD_WELD_DATA : WORD ;
    RBT3_STANDARD_WELD_DATA : WORD ;
    RBT4_STANDARD_WELD_DATA : WORD ;
    RBT5_STANDARD_WELD_DATA : WORD ;
    RBT6_STANDARD_WELD_DATA : WORD ;
    RBT7_STANDARD_WELD_DATA : WORD ;
    RBT8_STANDARD_WELD_DATA : WORD ;
    RBT9_STANDARD_WELD_DATA : WORD ;
    RBT10_STANDARD_WELD_DATA : WORD ;
    RBT11_STANDARD_WELD_DATA : WORD ;
    RBT12_STANDARD_WELD_DATA : WORD ;
    RBT13_STANDARD_WELD_DATA : WORD ;
    RBT14_STANDARD_WELD_DATA : WORD ;
    RBT15_STANDARD_WELD_DATA : WORD ;
    RBT16_STANDARD_WELD_DATA : WORD ;
    RBT17_STANDARD_WELD_DATA : WORD ;
    RBT18_STANDARD_WELD_DATA : WORD ;
    RBT19_STANDARD_WELD_DATA : WORD ;
    RBT20_STANDARD_WELD_DATA : WORD ;
    RBT21_STANDARD_WELD_DATA : WORD ;
    RBT22_STANDARD_WELD_DATA : WORD ;
    RBT23_STANDARD_WELD_DAT : WORD ;
    RBT24_STANDARD_WELD_DAT : WORD ;
    CHK_WORD : WORD ;
    TEST_TEMP : ARRAY  [1 .. 40 ] OF BYTE ;
   END_STRUCT ;
   S700_1_BT_CODE_2103 : STRUCT
    STATION_MAIN : WORD ;
    DISTINCTION_LH_RH : WORD ;
    STAION_NUMBER : WORD ;
    BODY_TYPE_1ST : WORD ;
    BODY_TYPE_OPTION : WORD ;
    RBT1_STANDARD_WELD_DATA : WORD ;
    RBT2_STANDARD_WELD_DATA : WORD ;
    RBT3_STANDARD_WELD_DATA : WORD ;
    RBT4_STANDARD_WELD_DATA : WORD ;
    RBT5_STANDARD_WELD_DATA : WORD ;
    RBT6_STANDARD_WELD_DATA : WORD ;
    RBT7_STANDARD_WELD_DATA : WORD ;
    RBT8_STANDARD_WELD_DATA : WORD ;
    RBT9_STANDARD_WELD_DATA : WORD ;
    RBT10_STANDARD_WELD_DATA : WORD ;
    RBT11_STANDARD_WELD_DATA : WORD ;
    RBT12_STANDARD_WELD_DATA : WORD ;
    RBT13_STANDARD_WELD_DATA : WORD ;
    RBT14_STANDARD_WELD_DATA : WORD ;
    RBT15_STANDARD_WELD_DATA : WORD ;
    RBT16_STANDARD_WELD_DATA : WORD ;
    RBT17_STANDARD_WELD_DATA : WORD ;
    RBT18_STANDARD_WELD_DATA : WORD ;
    RBT19_STANDARD_WELD_DATA : WORD ;
    RBT20_STANDARD_WELD_DATA : WORD ;
    RBT21_STANDARD_WELD_DATA : WORD ;
    RBT22_STANDARD_WELD_DATA : WORD ;
    RBT23_STANDARD_WELD_DAT : WORD ;
    RBT24_STANDARD_WELD_DAT : WORD ;
    CHK_WORD : WORD ;
    TEST_TEMP : ARRAY  [1 .. 40 ] OF BYTE ;
   END_STRUCT ;
   S700_1_BT_CODE_2104 : STRUCT
    STATION_MAIN : WORD ;
    DISTINCTION_LH_RH : WORD ;
    STAION_NUMBER : WORD ;
    BODY_TYPE_1ST : WORD ;
    BODY_TYPE_OPTION : WORD ;
    RBT1_STANDARD_WELD_DATA : WORD ;
    RBT2_STANDARD_WELD_DATA : WORD ;
    RBT3_STANDARD_WELD_DATA : WORD ;
    RBT4_STANDARD_WELD_DATA : WORD ;
    RBT5_STANDARD_WELD_DATA : WORD ;
    RBT6_STANDARD_WELD_DATA : WORD ;
    RBT7_STANDARD_WELD_DATA : WORD ;
    RBT8_STANDARD_WELD_DATA : WORD ;
    RBT9_STANDARD_WELD_DATA : WORD ;
    RBT10_STANDARD_WELD_DATA : WORD ;
    RBT11_STANDARD_WELD_DATA : WORD ;
    RBT12_STANDARD_WELD_DATA : WORD ;
    RBT13_STANDARD_WELD_DATA : WORD ;
    RBT14_STANDARD_WELD_DATA : WORD ;
    RBT15_STANDARD_WELD_DATA : WORD ;
    RBT16_STANDARD_WELD_DATA : WORD ;
    RBT17_STANDARD_WELD_DATA : WORD ;
    RBT18_STANDARD_WELD_DATA : WORD ;
    RBT19_STANDARD_WELD_DATA : WORD ;
    RBT20_STANDARD_WELD_DATA : WORD ;
    RBT21_STANDARD_WELD_DATA : WORD ;
    RBT22_STANDARD_WELD_DATA : WORD ;
    RBT23_STANDARD_WELD_DAT : WORD ;
    RBT24_STANDARD_WELD_DAT : WORD ;
    CHK_WORD : WORD ;
    TEST_TEMP : ARRAY  [1 .. 40 ] OF BYTE ;
   END_STRUCT ;
   S700_1_BT_CODE_2105 : STRUCT
    STATION_MAIN : WORD ;
    DISTINCTION_LH_RH : WORD ;
    STAION_NUMBER : WORD ;
    BODY_TYPE_1ST : WORD ;
    BODY_TYPE_OPTION : WORD ;
    RBT1_STANDARD_WELD_DATA : WORD ;
    RBT2_STANDARD_WELD_DATA : WORD ;
    RBT3_STANDARD_WELD_DATA : WORD ;
    RBT4_STANDARD_WELD_DATA : WORD ;
    RBT5_STANDARD_WELD_DATA : WORD ;
    RBT6_STANDARD_WELD_DATA : WORD ;
    RBT7_STANDARD_WELD_DATA : WORD ;
    RBT8_STANDARD_WELD_DATA : WORD ;
    RBT9_STANDARD_WELD_DATA : WORD ;
    RBT10_STANDARD_WELD_DATA : WORD ;
    RBT11_STANDARD_WELD_DATA : WORD ;
    RBT12_STANDARD_WELD_DATA : WORD ;
    RBT13_STANDARD_WELD_DATA : WORD ;
    RBT14_STANDARD_WELD_DATA : WORD ;
    RBT15_STANDARD_WELD_DATA : WORD ;
    RBT16_STANDARD_WELD_DATA : WORD ;
    RBT17_STANDARD_WELD_DATA : WORD ;
    RBT18_STANDARD_WELD_DATA : WORD ;
    RBT19_STANDARD_WELD_DATA : WORD ;
    RBT20_STANDARD_WELD_DATA : WORD ;
    RBT21_STANDARD_WELD_DATA : WORD ;
    RBT22_STANDARD_WELD_DATA : WORD ;
    RBT23_STANDARD_WELD_DAT : WORD ;
    RBT24_STANDARD_WELD_DAT : WORD ;
    CHK_WORD : WORD ;
    TEST_TEMP : ARRAY  [1 .. 40 ] OF BYTE ;
   END_STRUCT ;
   S700_1_BT_CODE_2106 : STRUCT
    STATION_MAIN : WORD ;
    DISTINCTION_LH_RH : WORD ;
    STAION_NUMBER : WORD ;
    BODY_TYPE_1ST : WORD ;
    BODY_TYPE_OPTION : WORD ;
    RBT1_STANDARD_WELD_DATA : WORD ;
    RBT2_STANDARD_WELD_DATA : WORD ;
    RBT3_STANDARD_WELD_DATA : WORD ;
    RBT4_STANDARD_WELD_DATA : WORD ;
    RBT5_STANDARD_WELD_DATA : WORD ;
    RBT6_STANDARD_WELD_DATA : WORD ;
    RBT7_STANDARD_WELD_DATA : WORD ;
    RBT8_STANDARD_WELD_DATA : WORD ;
    RBT9_STANDARD_WELD_DATA : WORD ;
    RBT10_STANDARD_WELD_DATA : WORD ;
    RBT11_STANDARD_WELD_DATA : WORD ;
    RBT12_STANDARD_WELD_DATA : WORD ;
    RBT13_STANDARD_WELD_DATA : WORD ;
    RBT14_STANDARD_WELD_DATA : WORD ;
    RBT15_STANDARD_WELD_DATA : WORD ;
    RBT16_STANDARD_WELD_DATA : WORD ;
    RBT17_STANDARD_WELD_DATA : WORD ;
    RBT18_STANDARD_WELD_DATA : WORD ;
    RBT19_STANDARD_WELD_DATA : WORD ;
    RBT20_STANDARD_WELD_DATA : WORD ;
    RBT21_STANDARD_WELD_DATA : WORD ;
    RBT22_STANDARD_WELD_DATA : WORD ;
    RBT23_STANDARD_WELD_DAT : WORD ;
    RBT24_STANDARD_WELD_DAT : WORD ;
    CHK_WORD : WORD ;
    TEST_TEMP : ARRAY  [1 .. 40 ] OF BYTE ;
   END_STRUCT ;
   S700_1_BT_CODE_2107 : STRUCT
    STATION_MAIN : WORD ;
    DISTINCTION_LH_RH : WORD ;
    STAION_NUMBER : WORD ;
    BODY_TYPE_1ST : WORD ;
    BODY_TYPE_OPTION : WORD ;
    RBT1_STANDARD_WELD_DATA : WORD ;
    RBT2_STANDARD_WELD_DATA : WORD ;
    RBT3_STANDARD_WELD_DATA : WORD ;
    RBT4_STANDARD_WELD_DATA : WORD ;
    RBT5_STANDARD_WELD_DATA : WORD ;
    RBT6_STANDARD_WELD_DATA : WORD ;
    RBT7_STANDARD_WELD_DATA : WORD ;
    RBT8_STANDARD_WELD_DATA : WORD ;
    RBT9_STANDARD_WELD_DATA : WORD ;
    RBT10_STANDARD_WELD_DATA : WORD ;
    RBT11_STANDARD_WELD_DATA : WORD ;
    RBT12_STANDARD_WELD_DATA : WORD ;
    RBT13_STANDARD_WELD_DATA : WORD ;
    RBT14_STANDARD_WELD_DATA : WORD ;
    RBT15_STANDARD_WELD_DATA : WORD ;
    RBT16_STANDARD_WELD_DATA : WORD ;
    RBT17_STANDARD_WELD_DATA : WORD ;
    RBT18_STANDARD_WELD_DATA : WORD ;
    RBT19_STANDARD_WELD_DATA : WORD ;
    RBT20_STANDARD_WELD_DATA : WORD ;
    RBT21_STANDARD_WELD_DATA : WORD ;
    RBT22_STANDARD_WELD_DATA : WORD ;
    RBT23_STANDARD_WELD_DAT : WORD ;
    RBT24_STANDARD_WELD_DAT : WORD ;
    CHK_WORD : WORD ;
    TEST_TEMP : ARRAY  [1 .. 40 ] OF BYTE ;
   END_STRUCT ;
   S700_1_BT_CODE_2108 : STRUCT
    STATION_MAIN : WORD ;
    DISTINCTION_LH_RH : WORD ;
    STAION_NUMBER : WORD ;
    BODY_TYPE_1ST : WORD ;
    BODY_TYPE_OPTION : WORD ;
    RBT1_STANDARD_WELD_DATA : WORD ;
    RBT2_STANDARD_WELD_DATA : WORD ;
    RBT3_STANDARD_WELD_DATA : WORD ;
    RBT4_STANDARD_WELD_DATA : WORD ;
    RBT5_STANDARD_WELD_DATA : WORD ;
    RBT6_STANDARD_WELD_DATA : WORD ;
    RBT7_STANDARD_WELD_DATA : WORD ;
    RBT8_STANDARD_WELD_DATA : WORD ;
    RBT9_STANDARD_WELD_DATA : WORD ;
    RBT10_STANDARD_WELD_DATA : WORD ;
    RBT11_STANDARD_WELD_DATA : WORD ;
    RBT12_STANDARD_WELD_DATA : WORD ;
    RBT13_STANDARD_WELD_DATA : WORD ;
    RBT14_STANDARD_WELD_DATA : WORD ;
    RBT15_STANDARD_WELD_DATA : WORD ;
    RBT16_STANDARD_WELD_DATA : WORD ;
    RBT17_STANDARD_WELD_DATA : WORD ;
    RBT18_STANDARD_WELD_DATA : WORD ;
    RBT19_STANDARD_WELD_DATA : WORD ;
    RBT20_STANDARD_WELD_DATA : WORD ;
    RBT21_STANDARD_WELD_DATA : WORD ;
    RBT22_STANDARD_WELD_DATA : WORD ;
    RBT23_STANDARD_WELD_DAT : WORD ;
    RBT24_STANDARD_WELD_DAT : WORD ;
    CHK_WORD : WORD ;
    TEST_TEMP : ARRAY  [1 .. 40 ] OF BYTE ;
   END_STRUCT ;
   S700_1_BT_CODE_2109 : STRUCT
    STATION_MAIN : WORD ;
    DISTINCTION_LH_RH : WORD ;
    STAION_NUMBER : WORD ;
    BODY_TYPE_1ST : WORD ;
    BODY_TYPE_OPTION : WORD ;
    RBT1_STANDARD_WELD_DATA : WORD ;
    RBT2_STANDARD_WELD_DATA : WORD ;
    RBT3_STANDARD_WELD_DATA : WORD ;
    RBT4_STANDARD_WELD_DATA : WORD ;
    RBT5_STANDARD_WELD_DATA : WORD ;
    RBT6_STANDARD_WELD_DATA : WORD ;
    RBT7_STANDARD_WELD_DATA : WORD ;
    RBT8_STANDARD_WELD_DATA : WORD ;
    RBT9_STANDARD_WELD_DATA : WORD ;
    RBT10_STANDARD_WELD_DATA : WORD ;
    RBT11_STANDARD_WELD_DATA : WORD ;
    RBT12_STANDARD_WELD_DATA : WORD ;
    RBT13_STANDARD_WELD_DATA : WORD ;
    RBT14_STANDARD_WELD_DATA : WORD ;
    RBT15_STANDARD_WELD_DATA : WORD ;
    RBT16_STANDARD_WELD_DATA : WORD ;
    RBT17_STANDARD_WELD_DATA : WORD ;
    RBT18_STANDARD_WELD_DATA : WORD ;
    RBT19_STANDARD_WELD_DATA : WORD ;
    RBT20_STANDARD_WELD_DATA : WORD ;
    RBT21_STANDARD_WELD_DATA : WORD ;
    RBT22_STANDARD_WELD_DATA : WORD ;
    RBT23_STANDARD_WELD_DAT : WORD ;
    RBT24_STANDARD_WELD_DAT : WORD ;
    CHK_WORD : WORD ;
    TEST_TEMP : ARRAY  [1 .. 40 ] OF BYTE ;
   END_STRUCT ;
   S700_1_BT_CODE_2110 : STRUCT
    STATION_MAIN : WORD ;
    DISTINCTION_LH_RH : WORD ;
    STAION_NUMBER : WORD ;
    BODY_TYPE_1ST : WORD ;
    BODY_TYPE_OPTION : WORD ;
    RBT1_STANDARD_WELD_DATA : WORD ;
    RBT2_STANDARD_WELD_DATA : WORD ;
    RBT3_STANDARD_WELD_DATA : WORD ;
    RBT4_STANDARD_WELD_DATA : WORD ;
    RBT5_STANDARD_WELD_DATA : WORD ;
    RBT6_STANDARD_WELD_DATA : WORD ;
    RBT7_STANDARD_WELD_DATA : WORD ;
    RBT8_STANDARD_WELD_DATA : WORD ;
    RBT9_STANDARD_WELD_DATA : WORD ;
    RBT10_STANDARD_WELD_DATA : WORD ;
    RBT11_STANDARD_WELD_DATA : WORD ;
    RBT12_STANDARD_WELD_DATA : WORD ;
    RBT13_STANDARD_WELD_DATA : WORD ;
    RBT14_STANDARD_WELD_DATA : WORD ;
    RBT15_STANDARD_WELD_DATA : WORD ;
    RBT16_STANDARD_WELD_DATA : WORD ;
    RBT17_STANDARD_WELD_DATA : WORD ;
    RBT18_STANDARD_WELD_DATA : WORD ;
    RBT19_STANDARD_WELD_DATA : WORD ;
    RBT20_STANDARD_WELD_DATA : WORD ;
    RBT21_STANDARD_WELD_DATA : WORD ;
    RBT22_STANDARD_WELD_DATA : WORD ;
    RBT23_STANDARD_WELD_DAT : WORD ;
    RBT24_STANDARD_WELD_DAT : WORD ;
    CHK_WORD : WORD ;
    TEST_TEMP : ARRAY  [1 .. 40 ] OF BYTE ;
   END_STRUCT ;
   S700_1_BT_CODE_2111 : STRUCT
    STATION_MAIN : WORD ;
    DISTINCTION_LH_RH : WORD ;
    STAION_NUMBER : WORD ;
    BODY_TYPE_1ST : WORD ;
    BODY_TYPE_OPTION : WORD ;
    RBT1_STANDARD_WELD_DATA : WORD ;
    RBT2_STANDARD_WELD_DATA : WORD ;
    RBT3_STANDARD_WELD_DATA : WORD ;
    RBT4_STANDARD_WELD_DATA : WORD ;
    RBT5_STANDARD_WELD_DATA : WORD ;
    RBT6_STANDARD_WELD_DATA : WORD ;
    RBT7_STANDARD_WELD_DATA : WORD ;
    RBT8_STANDARD_WELD_DATA : WORD ;
    RBT9_STANDARD_WELD_DATA : WORD ;
    RBT10_STANDARD_WELD_DATA : WORD ;
    RBT11_STANDARD_WELD_DATA : WORD ;
    RBT12_STANDARD_WELD_DATA : WORD ;
    RBT13_STANDARD_WELD_DATA : WORD ;
    RBT14_STANDARD_WELD_DATA : WORD ;
    RBT15_STANDARD_WELD_DATA : WORD ;
    RBT16_STANDARD_WELD_DATA : WORD ;
    RBT17_STANDARD_WELD_DATA : WORD ;
    RBT18_STANDARD_WELD_DATA : WORD ;
    RBT19_STANDARD_WELD_DATA : WORD ;
    RBT20_STANDARD_WELD_DATA : WORD ;
    RBT21_STANDARD_WELD_DATA : WORD ;
    RBT22_STANDARD_WELD_DATA : WORD ;
    RBT23_STANDARD_WELD_DAT : WORD ;
    RBT24_STANDARD_WELD_DAT : WORD ;
    CHK_WORD : WORD ;
    TEST_TEMP : ARRAY  [1 .. 40 ] OF BYTE ;
   END_STRUCT ;
   S700_1_BT_CODE_2112 : STRUCT
    STATION_MAIN : WORD ;
    DISTINCTION_LH_RH : WORD ;
    STAION_NUMBER : WORD ;
    BODY_TYPE_1ST : WORD ;
    BODY_TYPE_OPTION : WORD ;
    RBT1_STANDARD_WELD_DATA : WORD ;
    RBT2_STANDARD_WELD_DATA : WORD ;
    RBT3_STANDARD_WELD_DATA : WORD ;
    RBT4_STANDARD_WELD_DATA : WORD ;
    RBT5_STANDARD_WELD_DATA : WORD ;
    RBT6_STANDARD_WELD_DATA : WORD ;
    RBT7_STANDARD_WELD_DATA : WORD ;
    RBT8_STANDARD_WELD_DATA : WORD ;
    RBT9_STANDARD_WELD_DATA : WORD ;
    RBT10_STANDARD_WELD_DATA : WORD ;
    RBT11_STANDARD_WELD_DATA : WORD ;
    RBT12_STANDARD_WELD_DATA : WORD ;
    RBT13_STANDARD_WELD_DATA : WORD ;
    RBT14_STANDARD_WELD_DATA : WORD ;
    RBT15_STANDARD_WELD_DATA : WORD ;
    RBT16_STANDARD_WELD_DATA : WORD ;
    RBT17_STANDARD_WELD_DATA : WORD ;
    RBT18_STANDARD_WELD_DATA : WORD ;
    RBT19_STANDARD_WELD_DATA : WORD ;
    RBT20_STANDARD_WELD_DATA : WORD ;
    RBT21_STANDARD_WELD_DATA : WORD ;
    RBT22_STANDARD_WELD_DATA : WORD ;
    RBT23_STANDARD_WELD_DAT : WORD ;
    RBT24_STANDARD_WELD_DAT : WORD ;
    CHK_WORD : WORD ;
    TEST_TEMP : ARRAY  [1 .. 40 ] OF BYTE ;
   END_STRUCT ;
   S700_1_BT_CODE_2113 : STRUCT
    STATION_MAIN : WORD ;
    DISTINCTION_LH_RH : WORD ;
    STAION_NUMBER : WORD ;
    BODY_TYPE_1ST : WORD ;
    BODY_TYPE_OPTION : WORD ;
    RBT1_STANDARD_WELD_DATA : WORD ;
    RBT2_STANDARD_WELD_DATA : WORD ;
    RBT3_STANDARD_WELD_DATA : WORD ;
    RBT4_STANDARD_WELD_DATA : WORD ;
    RBT5_STANDARD_WELD_DATA : WORD ;
    RBT6_STANDARD_WELD_DATA : WORD ;
    RBT7_STANDARD_WELD_DATA : WORD ;
    RBT8_STANDARD_WELD_DATA : WORD ;
    RBT9_STANDARD_WELD_DATA : WORD ;
    RBT10_STANDARD_WELD_DATA : WORD ;
    RBT11_STANDARD_WELD_DATA : WORD ;
    RBT12_STANDARD_WELD_DATA : WORD ;
    RBT13_STANDARD_WELD_DATA : WORD ;
    RBT14_STANDARD_WELD_DATA : WORD ;
    RBT15_STANDARD_WELD_DATA : WORD ;
    RBT16_STANDARD_WELD_DATA : WORD ;
    RBT17_STANDARD_WELD_DATA : WORD ;
    RBT18_STANDARD_WELD_DATA : WORD ;
    RBT19_STANDARD_WELD_DATA : WORD ;
    RBT20_STANDARD_WELD_DATA : WORD ;
    RBT21_STANDARD_WELD_DATA : WORD ;
    RBT22_STANDARD_WELD_DATA : WORD ;
    RBT23_STANDARD_WELD_DAT : WORD ;
    RBT24_STANDARD_WELD_DAT : WORD ;
    CHK_WORD : WORD ;
    TEST_TEMP : ARRAY  [1 .. 40 ] OF BYTE ;
   END_STRUCT ;
   S700_1_BT_CODE_2114 : STRUCT
    STATION_MAIN : WORD ;
    DISTINCTION_LH_RH : WORD ;
    STAION_NUMBER : WORD ;
    BODY_TYPE_1ST : WORD ;
    BODY_TYPE_OPTION : WORD ;
    RBT1_STANDARD_WELD_DATA : WORD ;
    RBT2_STANDARD_WELD_DATA : WORD ;
    RBT3_STANDARD_WELD_DATA : WORD ;
    RBT4_STANDARD_WELD_DATA : WORD ;
    RBT5_STANDARD_WELD_DATA : WORD ;
    RBT6_STANDARD_WELD_DATA : WORD ;
    RBT7_STANDARD_WELD_DATA : WORD ;
    RBT8_STANDARD_WELD_DATA : WORD ;
    RBT9_STANDARD_WELD_DATA : WORD ;
    RBT10_STANDARD_WELD_DATA : WORD ;
    RBT11_STANDARD_WELD_DATA : WORD ;
    RBT12_STANDARD_WELD_DATA : WORD ;
    RBT13_STANDARD_WELD_DATA : WORD ;
    RBT14_STANDARD_WELD_DATA : WORD ;
    RBT15_STANDARD_WELD_DATA : WORD ;
    RBT16_STANDARD_WELD_DATA : WORD ;
    RBT17_STANDARD_WELD_DATA : WORD ;
    RBT18_STANDARD_WELD_DATA : WORD ;
    RBT19_STANDARD_WELD_DATA : WORD ;
    RBT20_STANDARD_WELD_DATA : WORD ;
    RBT21_STANDARD_WELD_DATA : WORD ;
    RBT22_STANDARD_WELD_DATA : WORD ;
    RBT23_STANDARD_WELD_DAT : WORD ;
    RBT24_STANDARD_WELD_DAT : WORD ;
    CHK_WORD : WORD ;
    TEST_TEMP : ARRAY  [1 .. 40 ] OF BYTE ;
   END_STRUCT ;
   S700_1_BT_CODE_2115 : STRUCT
    STATION_MAIN : WORD ;
    DISTINCTION_LH_RH : WORD ;
    STAION_NUMBER : WORD ;
    BODY_TYPE_1ST : WORD ;
    BODY_TYPE_OPTION : WORD ;
    RBT1_STANDARD_WELD_DATA : WORD ;
    RBT2_STANDARD_WELD_DATA : WORD ;
    RBT3_STANDARD_WELD_DATA : WORD ;
    RBT4_STANDARD_WELD_DATA : WORD ;
    RBT5_STANDARD_WELD_DATA : WORD ;
    RBT6_STANDARD_WELD_DATA : WORD ;
    RBT7_STANDARD_WELD_DATA : WORD ;
    RBT8_STANDARD_WELD_DATA : WORD ;
    RBT9_STANDARD_WELD_DATA : WORD ;
    RBT10_STANDARD_WELD_DATA : WORD ;
    RBT11_STANDARD_WELD_DATA : WORD ;
    RBT12_STANDARD_WELD_DATA : WORD ;
    RBT13_STANDARD_WELD_DATA : WORD ;
    RBT14_STANDARD_WELD_DATA : WORD ;
    RBT15_STANDARD_WELD_DATA : WORD ;
    RBT16_STANDARD_WELD_DATA : WORD ;
    RBT17_STANDARD_WELD_DATA : WORD ;
    RBT18_STANDARD_WELD_DATA : WORD ;
    RBT19_STANDARD_WELD_DATA : WORD ;
    RBT20_STANDARD_WELD_DATA : WORD ;
    RBT21_STANDARD_WELD_DATA : WORD ;
    RBT22_STANDARD_WELD_DATA : WORD ;
    RBT23_STANDARD_WELD_DAT : WORD ;
    RBT24_STANDARD_WELD_DAT : WORD ;
    CHK_WORD : WORD ;
    TEST_TEMP : ARRAY  [1 .. 40 ] OF BYTE ;
   END_STRUCT ;
   S700_1_BT_CODE_2116 : STRUCT
    STATION_MAIN : WORD ;
    DISTINCTION_LH_RH : WORD ;
    STAION_NUMBER : WORD ;
    BODY_TYPE_1ST : WORD ;
    BODY_TYPE_OPTION : WORD ;
    RBT1_STANDARD_WELD_DATA : WORD ;
    RBT2_STANDARD_WELD_DATA : WORD ;
    RBT3_STANDARD_WELD_DATA : WORD ;
    RBT4_STANDARD_WELD_DATA : WORD ;
    RBT5_STANDARD_WELD_DATA : WORD ;
    RBT6_STANDARD_WELD_DATA : WORD ;
    RBT7_STANDARD_WELD_DATA : WORD ;
    RBT8_STANDARD_WELD_DATA : WORD ;
    RBT9_STANDARD_WELD_DATA : WORD ;
    RBT10_STANDARD_WELD_DATA : WORD ;
    RBT11_STANDARD_WELD_DATA : WORD ;
    RBT12_STANDARD_WELD_DATA : WORD ;
    RBT13_STANDARD_WELD_DATA : WORD ;
    RBT14_STANDARD_WELD_DATA : WORD ;
    RBT15_STANDARD_WELD_DATA : WORD ;
    RBT16_STANDARD_WELD_DATA : WORD ;
    RBT17_STANDARD_WELD_DATA : WORD ;
    RBT18_STANDARD_WELD_DATA : WORD ;
    RBT19_STANDARD_WELD_DATA : WORD ;
    RBT20_STANDARD_WELD_DATA : WORD ;
    RBT21_STANDARD_WELD_DATA : WORD ;
    RBT22_STANDARD_WELD_DATA : WORD ;
    RBT23_STANDARD_WELD_DAT : WORD ;
    RBT24_STANDARD_WELD_DAT : WORD ;
    CHK_WORD : WORD ;
    TEST_TEMP : ARRAY  [1 .. 40 ] OF BYTE ;
   END_STRUCT ;
   S700_1_BT_CODE_2117 : STRUCT
    STATION_MAIN : WORD ;
    DISTINCTION_LH_RH : WORD ;
    STAION_NUMBER : WORD ;
    BODY_TYPE_1ST : WORD ;
    BODY_TYPE_OPTION : WORD ;
    RBT1_STANDARD_WELD_DATA : WORD ;
    RBT2_STANDARD_WELD_DATA : WORD ;
    RBT3_STANDARD_WELD_DATA : WORD ;
    RBT4_STANDARD_WELD_DATA : WORD ;
    RBT5_STANDARD_WELD_DATA : WORD ;
    RBT6_STANDARD_WELD_DATA : WORD ;
    RBT7_STANDARD_WELD_DATA : WORD ;
    RBT8_STANDARD_WELD_DATA : WORD ;
    RBT9_STANDARD_WELD_DATA : WORD ;
    RBT10_STANDARD_WELD_DATA : WORD ;
    RBT11_STANDARD_WELD_DATA : WORD ;
    RBT12_STANDARD_WELD_DATA : WORD ;
    RBT13_STANDARD_WELD_DATA : WORD ;
    RBT14_STANDARD_WELD_DATA : WORD ;
    RBT15_STANDARD_WELD_DATA : WORD ;
    RBT16_STANDARD_WELD_DATA : WORD ;
    RBT17_STANDARD_WELD_DATA : WORD ;
    RBT18_STANDARD_WELD_DATA : WORD ;
    RBT19_STANDARD_WELD_DATA : WORD ;
    RBT20_STANDARD_WELD_DATA : WORD ;
    RBT21_STANDARD_WELD_DATA : WORD ;
    RBT22_STANDARD_WELD_DATA : WORD ;
    RBT23_STANDARD_WELD_DAT : WORD ;
    RBT24_STANDARD_WELD_DAT : WORD ;
    CHK_WORD : WORD ;
    TEST_TEMP : ARRAY  [1 .. 40 ] OF BYTE ;
   END_STRUCT ;
   S700_1_BT_CODE_2118 : STRUCT
    STATION_MAIN : WORD ;
    DISTINCTION_LH_RH : WORD ;
    STAION_NUMBER : WORD ;
    BODY_TYPE_1ST : WORD ;
    BODY_TYPE_OPTION : WORD ;
    RBT1_STANDARD_WELD_DATA : WORD ;
    RBT2_STANDARD_WELD_DATA : WORD ;
    RBT3_STANDARD_WELD_DATA : WORD ;
    RBT4_STANDARD_WELD_DATA : WORD ;
    RBT5_STANDARD_WELD_DATA : WORD ;
    RBT6_STANDARD_WELD_DATA : WORD ;
    RBT7_STANDARD_WELD_DATA : WORD ;
    RBT8_STANDARD_WELD_DATA : WORD ;
    RBT9_STANDARD_WELD_DATA : WORD ;
    RBT10_STANDARD_WELD_DATA : WORD ;
    RBT11_STANDARD_WELD_DATA : WORD ;
    RBT12_STANDARD_WELD_DATA : WORD ;
    RBT13_STANDARD_WELD_DATA : WORD ;
    RBT14_STANDARD_WELD_DATA : WORD ;
    RBT15_STANDARD_WELD_DATA : WORD ;
    RBT16_STANDARD_WELD_DATA : WORD ;
    RBT17_STANDARD_WELD_DATA : WORD ;
    RBT18_STANDARD_WELD_DATA : WORD ;
    RBT19_STANDARD_WELD_DATA : WORD ;
    RBT20_STANDARD_WELD_DATA : WORD ;
    RBT21_STANDARD_WELD_DATA : WORD ;
    RBT22_STANDARD_WELD_DATA : WORD ;
    RBT23_STANDARD_WELD_DAT : WORD ;
    RBT24_STANDARD_WELD_DAT : WORD ;
    CHK_WORD : WORD ;
    TEST_TEMP : ARRAY  [1 .. 40 ] OF BYTE ;
   END_STRUCT ;
   S700_1_BT_CODE_2119 : STRUCT
    STATION_MAIN : WORD ;
    DISTINCTION_LH_RH : WORD ;
    STAION_NUMBER : WORD ;
    BODY_TYPE_1ST : WORD ;
    BODY_TYPE_OPTION : WORD ;
    RBT1_STANDARD_WELD_DATA : WORD ;
    RBT2_STANDARD_WELD_DATA : WORD ;
    RBT3_STANDARD_WELD_DATA : WORD ;
    RBT4_STANDARD_WELD_DATA : WORD ;
    RBT5_STANDARD_WELD_DATA : WORD ;
    RBT6_STANDARD_WELD_DATA : WORD ;
    RBT7_STANDARD_WELD_DATA : WORD ;
    RBT8_STANDARD_WELD_DATA : WORD ;
    RBT9_STANDARD_WELD_DATA : WORD ;
    RBT10_STANDARD_WELD_DATA : WORD ;
    RBT11_STANDARD_WELD_DATA : WORD ;
    RBT12_STANDARD_WELD_DATA : WORD ;
    RBT13_STANDARD_WELD_DATA : WORD ;
    RBT14_STANDARD_WELD_DATA : WORD ;
    RBT15_STANDARD_WELD_DATA : WORD ;
    RBT16_STANDARD_WELD_DATA : WORD ;
    RBT17_STANDARD_WELD_DATA : WORD ;
    RBT18_STANDARD_WELD_DATA : WORD ;
    RBT19_STANDARD_WELD_DATA : WORD ;
    RBT20_STANDARD_WELD_DATA : WORD ;
    RBT21_STANDARD_WELD_DATA : WORD ;
    RBT22_STANDARD_WELD_DATA : WORD ;
    RBT23_STANDARD_WELD_DAT : WORD ;
    RBT24_STANDARD_WELD_DAT : WORD ;
    CHK_WORD : WORD ;
    TEST_TEMP : ARRAY  [1 .. 40 ] OF BYTE ;
   END_STRUCT ;
   S700_1_BT_CODE_2120 : STRUCT
    STATION_MAIN : WORD ;
    DISTINCTION_LH_RH : WORD ;
    STAION_NUMBER : WORD ;
    BODY_TYPE_1ST : WORD ;
    BODY_TYPE_OPTION : WORD ;
    RBT1_STANDARD_WELD_DATA : WORD ;
    RBT2_STANDARD_WELD_DATA : WORD ;
    RBT3_STANDARD_WELD_DATA : WORD ;
    RBT4_STANDARD_WELD_DATA : WORD ;
    RBT5_STANDARD_WELD_DATA : WORD ;
    RBT6_STANDARD_WELD_DATA : WORD ;
    RBT7_STANDARD_WELD_DATA : WORD ;
    RBT8_STANDARD_WELD_DATA : WORD ;
    RBT9_STANDARD_WELD_DATA : WORD ;
    RBT10_STANDARD_WELD_DATA : WORD ;
    RBT11_STANDARD_WELD_DATA : WORD ;
    RBT12_STANDARD_WELD_DATA : WORD ;
    RBT13_STANDARD_WELD_DATA : WORD ;
    RBT14_STANDARD_WELD_DATA : WORD ;
    RBT15_STANDARD_WELD_DATA : WORD ;
    RBT16_STANDARD_WELD_DATA : WORD ;
    RBT17_STANDARD_WELD_DATA : WORD ;
    RBT18_STANDARD_WELD_DATA : WORD ;
    RBT19_STANDARD_WELD_DATA : WORD ;
    RBT20_STANDARD_WELD_DATA : WORD ;
    RBT21_STANDARD_WELD_DATA : WORD ;
    RBT22_STANDARD_WELD_DATA : WORD ;
    RBT23_STANDARD_WELD_DAT : WORD ;
    RBT24_STANDARD_WELD_DAT : WORD ;
    CHK_WORD : WORD ;
    TEST_TEMP : ARRAY  [1 .. 40 ] OF BYTE ;
   END_STRUCT ;
   S701_BT_CODE_2101 : STRUCT
    STATION_MAIN : WORD ;
    DISTINCTION_LH_RH : WORD ;
    STAION_NUMBER : WORD ;
    BODY_TYPE_1ST : WORD ;
    BODY_TYPE_OPTION : WORD ;
    RBT1_STANDARD_WELD_DATA : WORD ;
    RBT2_STANDARD_WELD_DATA : WORD ;
    RBT3_STANDARD_WELD_DATA : WORD ;
    RBT4_STANDARD_WELD_DATA : WORD ;
    RBT5_STANDARD_WELD_DATA : WORD ;
    RBT6_STANDARD_WELD_DATA : WORD ;
    RBT7_STANDARD_WELD_DATA : WORD ;
    RBT8_STANDARD_WELD_DATA : WORD ;
    RBT9_STANDARD_WELD_DATA : WORD ;
    RBT10_STANDARD_WELD_DATA : WORD ;
    RBT11_STANDARD_WELD_DATA : WORD ;
    RBT12_STANDARD_WELD_DATA : WORD ;
    RBT13_STANDARD_WELD_DATA : WORD ;
    RBT14_STANDARD_WELD_DATA : WORD ;
    RBT15_STANDARD_WELD_DATA : WORD ;
    RBT16_STANDARD_WELD_DATA : WORD ;
    RBT17_STANDARD_WELD_DATA : WORD ;
    RBT18_STANDARD_WELD_DATA : WORD ;
    RBT19_STANDARD_WELD_DATA : WORD ;
    RBT20_STANDARD_WELD_DATA : WORD ;
    RBT21_STANDARD_WELD_DATA : WORD ;
    RBT22_STANDARD_WELD_DATA : WORD ;
    RBT23_STANDARD_WELD_DAT : WORD ;
    RBT24_STANDARD_WELD_DAT : WORD ;
    CHK_WORD : WORD ;
    TEST_TEMP : ARRAY  [1 .. 40 ] OF BYTE ;
   END_STRUCT ;
   S701_BT_CODE_2102 : STRUCT
    STATION_MAIN : WORD ;
    DISTINCTION_LH_RH : WORD ;
    STAION_NUMBER : WORD ;
    BODY_TYPE_1ST : WORD ;
    BODY_TYPE_OPTION : WORD ;
    RBT1_STANDARD_WELD_DATA : WORD ;
    RBT2_STANDARD_WELD_DATA : WORD ;
    RBT3_STANDARD_WELD_DATA : WORD ;
    RBT4_STANDARD_WELD_DATA : WORD ;
    RBT5_STANDARD_WELD_DATA : WORD ;
    RBT6_STANDARD_WELD_DATA : WORD ;
    RBT7_STANDARD_WELD_DATA : WORD ;
    RBT8_STANDARD_WELD_DATA : WORD ;
    RBT9_STANDARD_WELD_DATA : WORD ;
    RBT10_STANDARD_WELD_DATA : WORD ;
    RBT11_STANDARD_WELD_DATA : WORD ;
    RBT12_STANDARD_WELD_DATA : WORD ;
    RBT13_STANDARD_WELD_DATA : WORD ;
    RBT14_STANDARD_WELD_DATA : WORD ;
    RBT15_STANDARD_WELD_DATA : WORD ;
    RBT16_STANDARD_WELD_DATA : WORD ;
    RBT17_STANDARD_WELD_DATA : WORD ;
    RBT18_STANDARD_WELD_DATA : WORD ;
    RBT19_STANDARD_WELD_DATA : WORD ;
    RBT20_STANDARD_WELD_DATA : WORD ;
    RBT21_STANDARD_WELD_DATA : WORD ;
    RBT22_STANDARD_WELD_DATA : WORD ;
    RBT23_STANDARD_WELD_DAT : WORD ;
    RBT24_STANDARD_WELD_DAT : WORD ;
    CHK_WORD : WORD ;
    TEST_TEMP : ARRAY  [1 .. 40 ] OF BYTE ;
   END_STRUCT ;
   S701_BT_CODE_2103 : STRUCT
    STATION_MAIN : WORD ;
    DISTINCTION_LH_RH : WORD ;
    STAION_NUMBER : WORD ;
    BODY_TYPE_1ST : WORD ;
    BODY_TYPE_OPTION : WORD ;
    RBT1_STANDARD_WELD_DATA : WORD ;
    RBT2_STANDARD_WELD_DATA : WORD ;
    RBT3_STANDARD_WELD_DATA : WORD ;
    RBT4_STANDARD_WELD_DATA : WORD ;
    RBT5_STANDARD_WELD_DATA : WORD ;
    RBT6_STANDARD_WELD_DATA : WORD ;
    RBT7_STANDARD_WELD_DATA : WORD ;
    RBT8_STANDARD_WELD_DATA : WORD ;
    RBT9_STANDARD_WELD_DATA : WORD ;
    RBT10_STANDARD_WELD_DATA : WORD ;
    RBT11_STANDARD_WELD_DATA : WORD ;
    RBT12_STANDARD_WELD_DATA : WORD ;
    RBT13_STANDARD_WELD_DATA : WORD ;
    RBT14_STANDARD_WELD_DATA : WORD ;
    RBT15_STANDARD_WELD_DATA : WORD ;
    RBT16_STANDARD_WELD_DATA : WORD ;
    RBT17_STANDARD_WELD_DATA : WORD ;
    RBT18_STANDARD_WELD_DATA : WORD ;
    RBT19_STANDARD_WELD_DATA : WORD ;
    RBT20_STANDARD_WELD_DATA : WORD ;
    RBT21_STANDARD_WELD_DATA : WORD ;
    RBT22_STANDARD_WELD_DATA : WORD ;
    RBT23_STANDARD_WELD_DAT : WORD ;
    RBT24_STANDARD_WELD_DAT : WORD ;
    CHK_WORD : WORD ;
    TEST_TEMP : ARRAY  [1 .. 40 ] OF BYTE ;
   END_STRUCT ;
   S701_BT_CODE_2104 : STRUCT
    STATION_MAIN : WORD ;
    DISTINCTION_LH_RH : WORD ;
    STAION_NUMBER : WORD ;
    BODY_TYPE_1ST : WORD ;
    BODY_TYPE_OPTION : WORD ;
    RBT1_STANDARD_WELD_DATA : WORD ;
    RBT2_STANDARD_WELD_DATA : WORD ;
    RBT3_STANDARD_WELD_DATA : WORD ;
    RBT4_STANDARD_WELD_DATA : WORD ;
    RBT5_STANDARD_WELD_DATA : WORD ;
    RBT6_STANDARD_WELD_DATA : WORD ;
    RBT7_STANDARD_WELD_DATA : WORD ;
    RBT8_STANDARD_WELD_DATA : WORD ;
    RBT9_STANDARD_WELD_DATA : WORD ;
    RBT10_STANDARD_WELD_DATA : WORD ;
    RBT11_STANDARD_WELD_DATA : WORD ;
    RBT12_STANDARD_WELD_DATA : WORD ;
    RBT13_STANDARD_WELD_DATA : WORD ;
    RBT14_STANDARD_WELD_DATA : WORD ;
    RBT15_STANDARD_WELD_DATA : WORD ;
    RBT16_STANDARD_WELD_DATA : WORD ;
    RBT17_STANDARD_WELD_DATA : WORD ;
    RBT18_STANDARD_WELD_DATA : WORD ;
    RBT19_STANDARD_WELD_DATA : WORD ;
    RBT20_STANDARD_WELD_DATA : WORD ;
    RBT21_STANDARD_WELD_DATA : WORD ;
    RBT22_STANDARD_WELD_DATA : WORD ;
    RBT23_STANDARD_WELD_DAT : WORD ;
    RBT24_STANDARD_WELD_DAT : WORD ;
    CHK_WORD : WORD ;
    TEST_TEMP : ARRAY  [1 .. 40 ] OF BYTE ;
   END_STRUCT ;
   S701_BT_CODE_2105 : STRUCT
    STATION_MAIN : WORD ;
    DISTINCTION_LH_RH : WORD ;
    STAION_NUMBER : WORD ;
    BODY_TYPE_1ST : WORD ;
    BODY_TYPE_OPTION : WORD ;
    RBT1_STANDARD_WELD_DATA : WORD ;
    RBT2_STANDARD_WELD_DATA : WORD ;
    RBT3_STANDARD_WELD_DATA : WORD ;
    RBT4_STANDARD_WELD_DATA : WORD ;
    RBT5_STANDARD_WELD_DATA : WORD ;
    RBT6_STANDARD_WELD_DATA : WORD ;
    RBT7_STANDARD_WELD_DATA : WORD ;
    RBT8_STANDARD_WELD_DATA : WORD ;
    RBT9_STANDARD_WELD_DATA : WORD ;
    RBT10_STANDARD_WELD_DATA : WORD ;
    RBT11_STANDARD_WELD_DATA : WORD ;
    RBT12_STANDARD_WELD_DATA : WORD ;
    RBT13_STANDARD_WELD_DATA : WORD ;
    RBT14_STANDARD_WELD_DATA : WORD ;
    RBT15_STANDARD_WELD_DATA : WORD ;
    RBT16_STANDARD_WELD_DATA : WORD ;
    RBT17_STANDARD_WELD_DATA : WORD ;
    RBT18_STANDARD_WELD_DATA : WORD ;
    RBT19_STANDARD_WELD_DATA : WORD ;
    RBT20_STANDARD_WELD_DATA : WORD ;
    RBT21_STANDARD_WELD_DATA : WORD ;
    RBT22_STANDARD_WELD_DATA : WORD ;
    RBT23_STANDARD_WELD_DAT : WORD ;
    RBT24_STANDARD_WELD_DAT : WORD ;
    CHK_WORD : WORD ;
    TEST_TEMP : ARRAY  [1 .. 40 ] OF BYTE ;
   END_STRUCT ;
   S701_BT_CODE_2106 : STRUCT
    STATION_MAIN : WORD ;
    DISTINCTION_LH_RH : WORD ;
    STAION_NUMBER : WORD ;
    BODY_TYPE_1ST : WORD ;
    BODY_TYPE_OPTION : WORD ;
    RBT1_STANDARD_WELD_DATA : WORD ;
    RBT2_STANDARD_WELD_DATA : WORD ;
    RBT3_STANDARD_WELD_DATA : WORD ;
    RBT4_STANDARD_WELD_DATA : WORD ;
    RBT5_STANDARD_WELD_DATA : WORD ;
    RBT6_STANDARD_WELD_DATA : WORD ;
    RBT7_STANDARD_WELD_DATA : WORD ;
    RBT8_STANDARD_WELD_DATA : WORD ;
    RBT9_STANDARD_WELD_DATA : WORD ;
    RBT10_STANDARD_WELD_DATA : WORD ;
    RBT11_STANDARD_WELD_DATA : WORD ;
    RBT12_STANDARD_WELD_DATA : WORD ;
    RBT13_STANDARD_WELD_DATA : WORD ;
    RBT14_STANDARD_WELD_DATA : WORD ;
    RBT15_STANDARD_WELD_DATA : WORD ;
    RBT16_STANDARD_WELD_DATA : WORD ;
    RBT17_STANDARD_WELD_DATA : WORD ;
    RBT18_STANDARD_WELD_DATA : WORD ;
    RBT19_STANDARD_WELD_DATA : WORD ;
    RBT20_STANDARD_WELD_DATA : WORD ;
    RBT21_STANDARD_WELD_DATA : WORD ;
    RBT22_STANDARD_WELD_DATA : WORD ;
    RBT23_STANDARD_WELD_DAT : WORD ;
    RBT24_STANDARD_WELD_DAT : WORD ;
    CHK_WORD : WORD ;
    TEST_TEMP : ARRAY  [1 .. 40 ] OF BYTE ;
   END_STRUCT ;
   S701_BT_CODE_2107 : STRUCT
    STATION_MAIN : WORD ;
    DISTINCTION_LH_RH : WORD ;
    STAION_NUMBER : WORD ;
    BODY_TYPE_1ST : WORD ;
    BODY_TYPE_OPTION : WORD ;
    RBT1_STANDARD_WELD_DATA : WORD ;
    RBT2_STANDARD_WELD_DATA : WORD ;
    RBT3_STANDARD_WELD_DATA : WORD ;
    RBT4_STANDARD_WELD_DATA : WORD ;
    RBT5_STANDARD_WELD_DATA : WORD ;
    RBT6_STANDARD_WELD_DATA : WORD ;
    RBT7_STANDARD_WELD_DATA : WORD ;
    RBT8_STANDARD_WELD_DATA : WORD ;
    RBT9_STANDARD_WELD_DATA : WORD ;
    RBT10_STANDARD_WELD_DATA : WORD ;
    RBT11_STANDARD_WELD_DATA : WORD ;
    RBT12_STANDARD_WELD_DATA : WORD ;
    RBT13_STANDARD_WELD_DATA : WORD ;
    RBT14_STANDARD_WELD_DATA : WORD ;
    RBT15_STANDARD_WELD_DATA : WORD ;
    RBT16_STANDARD_WELD_DATA : WORD ;
    RBT17_STANDARD_WELD_DATA : WORD ;
    RBT18_STANDARD_WELD_DATA : WORD ;
    RBT19_STANDARD_WELD_DATA : WORD ;
    RBT20_STANDARD_WELD_DATA : WORD ;
    RBT21_STANDARD_WELD_DATA : WORD ;
    RBT22_STANDARD_WELD_DATA : WORD ;
    RBT23_STANDARD_WELD_DAT : WORD ;
    RBT24_STANDARD_WELD_DAT : WORD ;
    CHK_WORD : WORD ;
    TEST_TEMP : ARRAY  [1 .. 40 ] OF BYTE ;
   END_STRUCT ;
   S701_BT_CODE_2108 : STRUCT
    STATION_MAIN : WORD ;
    DISTINCTION_LH_RH : WORD ;
    STAION_NUMBER : WORD ;
    BODY_TYPE_1ST : WORD ;
    BODY_TYPE_OPTION : WORD ;
    RBT1_STANDARD_WELD_DATA : WORD ;
    RBT2_STANDARD_WELD_DATA : WORD ;
    RBT3_STANDARD_WELD_DATA : WORD ;
    RBT4_STANDARD_WELD_DATA : WORD ;
    RBT5_STANDARD_WELD_DATA : WORD ;
    RBT6_STANDARD_WELD_DATA : WORD ;
    RBT7_STANDARD_WELD_DATA : WORD ;
    RBT8_STANDARD_WELD_DATA : WORD ;
    RBT9_STANDARD_WELD_DATA : WORD ;
    RBT10_STANDARD_WELD_DATA : WORD ;
    RBT11_STANDARD_WELD_DATA : WORD ;
    RBT12_STANDARD_WELD_DATA : WORD ;
    RBT13_STANDARD_WELD_DATA : WORD ;
    RBT14_STANDARD_WELD_DATA : WORD ;
    RBT15_STANDARD_WELD_DATA : WORD ;
    RBT16_STANDARD_WELD_DATA : WORD ;
    RBT17_STANDARD_WELD_DATA : WORD ;
    RBT18_STANDARD_WELD_DATA : WORD ;
    RBT19_STANDARD_WELD_DATA : WORD ;
    RBT20_STANDARD_WELD_DATA : WORD ;
    RBT21_STANDARD_WELD_DATA : WORD ;
    RBT22_STANDARD_WELD_DATA : WORD ;
    RBT23_STANDARD_WELD_DAT : WORD ;
    RBT24_STANDARD_WELD_DAT : WORD ;
    CHK_WORD : WORD ;
    TEST_TEMP : ARRAY  [1 .. 40 ] OF BYTE ;
   END_STRUCT ;
   S701_BT_CODE_2109 : STRUCT
    STATION_MAIN : WORD ;
    DISTINCTION_LH_RH : WORD ;
    STAION_NUMBER : WORD ;
    BODY_TYPE_1ST : WORD ;
    BODY_TYPE_OPTION : WORD ;
    RBT1_STANDARD_WELD_DATA : WORD ;
    RBT2_STANDARD_WELD_DATA : WORD ;
    RBT3_STANDARD_WELD_DATA : WORD ;
    RBT4_STANDARD_WELD_DATA : WORD ;
    RBT5_STANDARD_WELD_DATA : WORD ;
    RBT6_STANDARD_WELD_DATA : WORD ;
    RBT7_STANDARD_WELD_DATA : WORD ;
    RBT8_STANDARD_WELD_DATA : WORD ;
    RBT9_STANDARD_WELD_DATA : WORD ;
    RBT10_STANDARD_WELD_DATA : WORD ;
    RBT11_STANDARD_WELD_DATA : WORD ;
    RBT12_STANDARD_WELD_DATA : WORD ;
    RBT13_STANDARD_WELD_DATA : WORD ;
    RBT14_STANDARD_WELD_DATA : WORD ;
    RBT15_STANDARD_WELD_DATA : WORD ;
    RBT16_STANDARD_WELD_DATA : WORD ;
    RBT17_STANDARD_WELD_DATA : WORD ;
    RBT18_STANDARD_WELD_DATA : WORD ;
    RBT19_STANDARD_WELD_DATA : WORD ;
    RBT20_STANDARD_WELD_DATA : WORD ;
    RBT21_STANDARD_WELD_DATA : WORD ;
    RBT22_STANDARD_WELD_DATA : WORD ;
    RBT23_STANDARD_WELD_DAT : WORD ;
    RBT24_STANDARD_WELD_DAT : WORD ;
    CHK_WORD : WORD ;
    TEST_TEMP : ARRAY  [1 .. 40 ] OF BYTE ;
   END_STRUCT ;
   S701_BT_CODE_2110 : STRUCT
    STATION_MAIN : WORD ;
    DISTINCTION_LH_RH : WORD ;
    STAION_NUMBER : WORD ;
    BODY_TYPE_1ST : WORD ;
    BODY_TYPE_OPTION : WORD ;
    RBT1_STANDARD_WELD_DATA : WORD ;
    RBT2_STANDARD_WELD_DATA : WORD ;
    RBT3_STANDARD_WELD_DATA : WORD ;
    RBT4_STANDARD_WELD_DATA : WORD ;
    RBT5_STANDARD_WELD_DATA : WORD ;
    RBT6_STANDARD_WELD_DATA : WORD ;
    RBT7_STANDARD_WELD_DATA : WORD ;
    RBT8_STANDARD_WELD_DATA : WORD ;
    RBT9_STANDARD_WELD_DATA : WORD ;
    RBT10_STANDARD_WELD_DATA : WORD ;
    RBT11_STANDARD_WELD_DATA : WORD ;
    RBT12_STANDARD_WELD_DATA : WORD ;
    RBT13_STANDARD_WELD_DATA : WORD ;
    RBT14_STANDARD_WELD_DATA : WORD ;
    RBT15_STANDARD_WELD_DATA : WORD ;
    RBT16_STANDARD_WELD_DATA : WORD ;
    RBT17_STANDARD_WELD_DATA : WORD ;
    RBT18_STANDARD_WELD_DATA : WORD ;
    RBT19_STANDARD_WELD_DATA : WORD ;
    RBT20_STANDARD_WELD_DATA : WORD ;
    RBT21_STANDARD_WELD_DATA : WORD ;
    RBT22_STANDARD_WELD_DATA : WORD ;
    RBT23_STANDARD_WELD_DAT : WORD ;
    RBT24_STANDARD_WELD_DAT : WORD ;
    CHK_WORD : WORD ;
    TEST_TEMP : ARRAY  [1 .. 40 ] OF BYTE ;
   END_STRUCT ;
   S701_BT_CODE_2111 : STRUCT
    STATION_MAIN : WORD ;
    DISTINCTION_LH_RH : WORD ;
    STAION_NUMBER : WORD ;
    BODY_TYPE_1ST : WORD ;
    BODY_TYPE_OPTION : WORD ;
    RBT1_STANDARD_WELD_DATA : WORD ;
    RBT2_STANDARD_WELD_DATA : WORD ;
    RBT3_STANDARD_WELD_DATA : WORD ;
    RBT4_STANDARD_WELD_DATA : WORD ;
    RBT5_STANDARD_WELD_DATA : WORD ;
    RBT6_STANDARD_WELD_DATA : WORD ;
    RBT7_STANDARD_WELD_DATA : WORD ;
    RBT8_STANDARD_WELD_DATA : WORD ;
    RBT9_STANDARD_WELD_DATA : WORD ;
    RBT10_STANDARD_WELD_DATA : WORD ;
    RBT11_STANDARD_WELD_DATA : WORD ;
    RBT12_STANDARD_WELD_DATA : WORD ;
    RBT13_STANDARD_WELD_DATA : WORD ;
    RBT14_STANDARD_WELD_DATA : WORD ;
    RBT15_STANDARD_WELD_DATA : WORD ;
    RBT16_STANDARD_WELD_DATA : WORD ;
    RBT17_STANDARD_WELD_DATA : WORD ;
    RBT18_STANDARD_WELD_DATA : WORD ;
    RBT19_STANDARD_WELD_DATA : WORD ;
    RBT20_STANDARD_WELD_DATA : WORD ;
    RBT21_STANDARD_WELD_DATA : WORD ;
    RBT22_STANDARD_WELD_DATA : WORD ;
    RBT23_STANDARD_WELD_DAT : WORD ;
    RBT24_STANDARD_WELD_DAT : WORD ;
    CHK_WORD : WORD ;
    TEST_TEMP : ARRAY  [1 .. 40 ] OF BYTE ;
   END_STRUCT ;
   S701_BT_CODE_2112 : STRUCT
    STATION_MAIN : WORD ;
    DISTINCTION_LH_RH : WORD ;
    STAION_NUMBER : WORD ;
    BODY_TYPE_1ST : WORD ;
    BODY_TYPE_OPTION : WORD ;
    RBT1_STANDARD_WELD_DATA : WORD ;
    RBT2_STANDARD_WELD_DATA : WORD ;
    RBT3_STANDARD_WELD_DATA : WORD ;
    RBT4_STANDARD_WELD_DATA : WORD ;
    RBT5_STANDARD_WELD_DATA : WORD ;
    RBT6_STANDARD_WELD_DATA : WORD ;
    RBT7_STANDARD_WELD_DATA : WORD ;
    RBT8_STANDARD_WELD_DATA : WORD ;
    RBT9_STANDARD_WELD_DATA : WORD ;
    RBT10_STANDARD_WELD_DATA : WORD ;
    RBT11_STANDARD_WELD_DATA : WORD ;
    RBT12_STANDARD_WELD_DATA : WORD ;
    RBT13_STANDARD_WELD_DATA : WORD ;
    RBT14_STANDARD_WELD_DATA : WORD ;
    RBT15_STANDARD_WELD_DATA : WORD ;
    RBT16_STANDARD_WELD_DATA : WORD ;
    RBT17_STANDARD_WELD_DATA : WORD ;
    RBT18_STANDARD_WELD_DATA : WORD ;
    RBT19_STANDARD_WELD_DATA : WORD ;
    RBT20_STANDARD_WELD_DATA : WORD ;
    RBT21_STANDARD_WELD_DATA : WORD ;
    RBT22_STANDARD_WELD_DATA : WORD ;
    RBT23_STANDARD_WELD_DAT : WORD ;
    RBT24_STANDARD_WELD_DAT : WORD ;
    CHK_WORD : WORD ;
    TEST_TEMP : ARRAY  [1 .. 40 ] OF BYTE ;
   END_STRUCT ;
   S701_BT_CODE_2113 : STRUCT
    STATION_MAIN : WORD ;
    DISTINCTION_LH_RH : WORD ;
    STAION_NUMBER : WORD ;
    BODY_TYPE_1ST : WORD ;
    BODY_TYPE_OPTION : WORD ;
    RBT1_STANDARD_WELD_DATA : WORD ;
    RBT2_STANDARD_WELD_DATA : WORD ;
    RBT3_STANDARD_WELD_DATA : WORD ;
    RBT4_STANDARD_WELD_DATA : WORD ;
    RBT5_STANDARD_WELD_DATA : WORD ;
    RBT6_STANDARD_WELD_DATA : WORD ;
    RBT7_STANDARD_WELD_DATA : WORD ;
    RBT8_STANDARD_WELD_DATA : WORD ;
    RBT9_STANDARD_WELD_DATA : WORD ;
    RBT10_STANDARD_WELD_DATA : WORD ;
    RBT11_STANDARD_WELD_DATA : WORD ;
    RBT12_STANDARD_WELD_DATA : WORD ;
    RBT13_STANDARD_WELD_DATA : WORD ;
    RBT14_STANDARD_WELD_DATA : WORD ;
    RBT15_STANDARD_WELD_DATA : WORD ;
    RBT16_STANDARD_WELD_DATA : WORD ;
    RBT17_STANDARD_WELD_DATA : WORD ;
    RBT18_STANDARD_WELD_DATA : WORD ;
    RBT19_STANDARD_WELD_DATA : WORD ;
    RBT20_STANDARD_WELD_DATA : WORD ;
    RBT21_STANDARD_WELD_DATA : WORD ;
    RBT22_STANDARD_WELD_DATA : WORD ;
    RBT23_STANDARD_WELD_DAT : WORD ;
    RBT24_STANDARD_WELD_DAT : WORD ;
    CHK_WORD : WORD ;
    TEST_TEMP : ARRAY  [1 .. 40 ] OF BYTE ;
   END_STRUCT ;
   S701_BT_CODE_2114 : STRUCT
    STATION_MAIN : WORD ;
    DISTINCTION_LH_RH : WORD ;
    STAION_NUMBER : WORD ;
    BODY_TYPE_1ST : WORD ;
    BODY_TYPE_OPTION : WORD ;
    RBT1_STANDARD_WELD_DATA : WORD ;
    RBT2_STANDARD_WELD_DATA : WORD ;
    RBT3_STANDARD_WELD_DATA : WORD ;
    RBT4_STANDARD_WELD_DATA : WORD ;
    RBT5_STANDARD_WELD_DATA : WORD ;
    RBT6_STANDARD_WELD_DATA : WORD ;
    RBT7_STANDARD_WELD_DATA : WORD ;
    RBT8_STANDARD_WELD_DATA : WORD ;
    RBT9_STANDARD_WELD_DATA : WORD ;
    RBT10_STANDARD_WELD_DATA : WORD ;
    RBT11_STANDARD_WELD_DATA : WORD ;
    RBT12_STANDARD_WELD_DATA : WORD ;
    RBT13_STANDARD_WELD_DATA : WORD ;
    RBT14_STANDARD_WELD_DATA : WORD ;
    RBT15_STANDARD_WELD_DATA : WORD ;
    RBT16_STANDARD_WELD_DATA : WORD ;
    RBT17_STANDARD_WELD_DATA : WORD ;
    RBT18_STANDARD_WELD_DATA : WORD ;
    RBT19_STANDARD_WELD_DATA : WORD ;
    RBT20_STANDARD_WELD_DATA : WORD ;
    RBT21_STANDARD_WELD_DATA : WORD ;
    RBT22_STANDARD_WELD_DATA : WORD ;
    RBT23_STANDARD_WELD_DAT : WORD ;
    RBT24_STANDARD_WELD_DAT : WORD ;
    CHK_WORD : WORD ;
    TEST_TEMP : ARRAY  [1 .. 40 ] OF BYTE ;
   END_STRUCT ;
   S701_BT_CODE_2115 : STRUCT
    STATION_MAIN : WORD ;
    DISTINCTION_LH_RH : WORD ;
    STAION_NUMBER : WORD ;
    BODY_TYPE_1ST : WORD ;
    BODY_TYPE_OPTION : WORD ;
    RBT1_STANDARD_WELD_DATA : WORD ;
    RBT2_STANDARD_WELD_DATA : WORD ;
    RBT3_STANDARD_WELD_DATA : WORD ;
    RBT4_STANDARD_WELD_DATA : WORD ;
    RBT5_STANDARD_WELD_DATA : WORD ;
    RBT6_STANDARD_WELD_DATA : WORD ;
    RBT7_STANDARD_WELD_DATA : WORD ;
    RBT8_STANDARD_WELD_DATA : WORD ;
    RBT9_STANDARD_WELD_DATA : WORD ;
    RBT10_STANDARD_WELD_DATA : WORD ;
    RBT11_STANDARD_WELD_DATA : WORD ;
    RBT12_STANDARD_WELD_DATA : WORD ;
    RBT13_STANDARD_WELD_DATA : WORD ;
    RBT14_STANDARD_WELD_DATA : WORD ;
    RBT15_STANDARD_WELD_DATA : WORD ;
    RBT16_STANDARD_WELD_DATA : WORD ;
    RBT17_STANDARD_WELD_DATA : WORD ;
    RBT18_STANDARD_WELD_DATA : WORD ;
    RBT19_STANDARD_WELD_DATA : WORD ;
    RBT20_STANDARD_WELD_DATA : WORD ;
    RBT21_STANDARD_WELD_DATA : WORD ;
    RBT22_STANDARD_WELD_DATA : WORD ;
    RBT23_STANDARD_WELD_DAT : WORD ;
    RBT24_STANDARD_WELD_DAT : WORD ;
    CHK_WORD : WORD ;
    TEST_TEMP : ARRAY  [1 .. 40 ] OF BYTE ;
   END_STRUCT ;
   S701_BT_CODE_2116 : STRUCT
    STATION_MAIN : WORD ;
    DISTINCTION_LH_RH : WORD ;
    STAION_NUMBER : WORD ;
    BODY_TYPE_1ST : WORD ;
    BODY_TYPE_OPTION : WORD ;
    RBT1_STANDARD_WELD_DATA : WORD ;
    RBT2_STANDARD_WELD_DATA : WORD ;
    RBT3_STANDARD_WELD_DATA : WORD ;
    RBT4_STANDARD_WELD_DATA : WORD ;
    RBT5_STANDARD_WELD_DATA : WORD ;
    RBT6_STANDARD_WELD_DATA : WORD ;
    RBT7_STANDARD_WELD_DATA : WORD ;
    RBT8_STANDARD_WELD_DATA : WORD ;
    RBT9_STANDARD_WELD_DATA : WORD ;
    RBT10_STANDARD_WELD_DATA : WORD ;
    RBT11_STANDARD_WELD_DATA : WORD ;
    RBT12_STANDARD_WELD_DATA : WORD ;
    RBT13_STANDARD_WELD_DATA : WORD ;
    RBT14_STANDARD_WELD_DATA : WORD ;
    RBT15_STANDARD_WELD_DATA : WORD ;
    RBT16_STANDARD_WELD_DATA : WORD ;
    RBT17_STANDARD_WELD_DATA : WORD ;
    RBT18_STANDARD_WELD_DATA : WORD ;
    RBT19_STANDARD_WELD_DATA : WORD ;
    RBT20_STANDARD_WELD_DATA : WORD ;
    RBT21_STANDARD_WELD_DATA : WORD ;
    RBT22_STANDARD_WELD_DATA : WORD ;
    RBT23_STANDARD_WELD_DAT : WORD ;
    RBT24_STANDARD_WELD_DAT : WORD ;
    CHK_WORD : WORD ;
    TEST_TEMP : ARRAY  [1 .. 40 ] OF BYTE ;
   END_STRUCT ;
   S701_BT_CODE_2117 : STRUCT
    STATION_MAIN : WORD ;
    DISTINCTION_LH_RH : WORD ;
    STAION_NUMBER : WORD ;
    BODY_TYPE_1ST : WORD ;
    BODY_TYPE_OPTION : WORD ;
    RBT1_STANDARD_WELD_DATA : WORD ;
    RBT2_STANDARD_WELD_DATA : WORD ;
    RBT3_STANDARD_WELD_DATA : WORD ;
    RBT4_STANDARD_WELD_DATA : WORD ;
    RBT5_STANDARD_WELD_DATA : WORD ;
    RBT6_STANDARD_WELD_DATA : WORD ;
    RBT7_STANDARD_WELD_DATA : WORD ;
    RBT8_STANDARD_WELD_DATA : WORD ;
    RBT9_STANDARD_WELD_DATA : WORD ;
    RBT10_STANDARD_WELD_DATA : WORD ;
    RBT11_STANDARD_WELD_DATA : WORD ;
    RBT12_STANDARD_WELD_DATA : WORD ;
    RBT13_STANDARD_WELD_DATA : WORD ;
    RBT14_STANDARD_WELD_DATA : WORD ;
    RBT15_STANDARD_WELD_DATA : WORD ;
    RBT16_STANDARD_WELD_DATA : WORD ;
    RBT17_STANDARD_WELD_DATA : WORD ;
    RBT18_STANDARD_WELD_DATA : WORD ;
    RBT19_STANDARD_WELD_DATA : WORD ;
    RBT20_STANDARD_WELD_DATA : WORD ;
    RBT21_STANDARD_WELD_DATA : WORD ;
    RBT22_STANDARD_WELD_DATA : WORD ;
    RBT23_STANDARD_WELD_DAT : WORD ;
    RBT24_STANDARD_WELD_DAT : WORD ;
    CHK_WORD : WORD ;
    TEST_TEMP : ARRAY  [1 .. 40 ] OF BYTE ;
   END_STRUCT ;
   S701_BT_CODE_2118 : STRUCT
    STATION_MAIN : WORD ;
    DISTINCTION_LH_RH : WORD ;
    STAION_NUMBER : WORD ;
    BODY_TYPE_1ST : WORD ;
    BODY_TYPE_OPTION : WORD ;
    RBT1_STANDARD_WELD_DATA : WORD ;
    RBT2_STANDARD_WELD_DATA : WORD ;
    RBT3_STANDARD_WELD_DATA : WORD ;
    RBT4_STANDARD_WELD_DATA : WORD ;
    RBT5_STANDARD_WELD_DATA : WORD ;
    RBT6_STANDARD_WELD_DATA : WORD ;
    RBT7_STANDARD_WELD_DATA : WORD ;
    RBT8_STANDARD_WELD_DATA : WORD ;
    RBT9_STANDARD_WELD_DATA : WORD ;
    RBT10_STANDARD_WELD_DATA : WORD ;
    RBT11_STANDARD_WELD_DATA : WORD ;
    RBT12_STANDARD_WELD_DATA : WORD ;
    RBT13_STANDARD_WELD_DATA : WORD ;
    RBT14_STANDARD_WELD_DATA : WORD ;
    RBT15_STANDARD_WELD_DATA : WORD ;
    RBT16_STANDARD_WELD_DATA : WORD ;
    RBT17_STANDARD_WELD_DATA : WORD ;
    RBT18_STANDARD_WELD_DATA : WORD ;
    RBT19_STANDARD_WELD_DATA : WORD ;
    RBT20_STANDARD_WELD_DATA : WORD ;
    RBT21_STANDARD_WELD_DATA : WORD ;
    RBT22_STANDARD_WELD_DATA : WORD ;
    RBT23_STANDARD_WELD_DAT : WORD ;
    RBT24_STANDARD_WELD_DAT : WORD ;
    CHK_WORD : WORD ;
    TEST_TEMP : ARRAY  [1 .. 40 ] OF BYTE ;
   END_STRUCT ;
   S701_BT_CODE_2119 : STRUCT
    STATION_MAIN : WORD ;
    DISTINCTION_LH_RH : WORD ;
    STAION_NUMBER : WORD ;
    BODY_TYPE_1ST : WORD ;
    BODY_TYPE_OPTION : WORD ;
    RBT1_STANDARD_WELD_DATA : WORD ;
    RBT2_STANDARD_WELD_DATA : WORD ;
    RBT3_STANDARD_WELD_DATA : WORD ;
    RBT4_STANDARD_WELD_DATA : WORD ;
    RBT5_STANDARD_WELD_DATA : WORD ;
    RBT6_STANDARD_WELD_DATA : WORD ;
    RBT7_STANDARD_WELD_DATA : WORD ;
    RBT8_STANDARD_WELD_DATA : WORD ;
    RBT9_STANDARD_WELD_DATA : WORD ;
    RBT10_STANDARD_WELD_DATA : WORD ;
    RBT11_STANDARD_WELD_DATA : WORD ;
    RBT12_STANDARD_WELD_DATA : WORD ;
    RBT13_STANDARD_WELD_DATA : WORD ;
    RBT14_STANDARD_WELD_DATA : WORD ;
    RBT15_STANDARD_WELD_DATA : WORD ;
    RBT16_STANDARD_WELD_DATA : WORD ;
    RBT17_STANDARD_WELD_DATA : WORD ;
    RBT18_STANDARD_WELD_DATA : WORD ;
    RBT19_STANDARD_WELD_DATA : WORD ;
    RBT20_STANDARD_WELD_DATA : WORD ;
    RBT21_STANDARD_WELD_DATA : WORD ;
    RBT22_STANDARD_WELD_DATA : WORD ;
    RBT23_STANDARD_WELD_DAT : WORD ;
    RBT24_STANDARD_WELD_DAT : WORD ;
    CHK_WORD : WORD ;
    TEST_TEMP : ARRAY  [1 .. 40 ] OF BYTE ;
   END_STRUCT ;
   S701_BT_CODE_2120 : STRUCT
    STATION_MAIN : WORD ;
    DISTINCTION_LH_RH : WORD ;
    STAION_NUMBER : WORD ;
    BODY_TYPE_1ST : WORD ;
    BODY_TYPE_OPTION : WORD ;
    RBT1_STANDARD_WELD_DATA : WORD ;
    RBT2_STANDARD_WELD_DATA : WORD ;
    RBT3_STANDARD_WELD_DATA : WORD ;
    RBT4_STANDARD_WELD_DATA : WORD ;
    RBT5_STANDARD_WELD_DATA : WORD ;
    RBT6_STANDARD_WELD_DATA : WORD ;
    RBT7_STANDARD_WELD_DATA : WORD ;
    RBT8_STANDARD_WELD_DATA : WORD ;
    RBT9_STANDARD_WELD_DATA : WORD ;
    RBT10_STANDARD_WELD_DATA : WORD ;
    RBT11_STANDARD_WELD_DATA : WORD ;
    RBT12_STANDARD_WELD_DATA : WORD ;
    RBT13_STANDARD_WELD_DATA : WORD ;
    RBT14_STANDARD_WELD_DATA : WORD ;
    RBT15_STANDARD_WELD_DATA : WORD ;
    RBT16_STANDARD_WELD_DATA : WORD ;
    RBT17_STANDARD_WELD_DATA : WORD ;
    RBT18_STANDARD_WELD_DATA : WORD ;
    RBT19_STANDARD_WELD_DATA : WORD ;
    RBT20_STANDARD_WELD_DATA : WORD ;
    RBT21_STANDARD_WELD_DATA : WORD ;
    RBT22_STANDARD_WELD_DATA : WORD ;
    RBT23_STANDARD_WELD_DAT : WORD ;
    RBT24_STANDARD_WELD_DAT : WORD ;
    CHK_WORD : WORD ;
    TEST_TEMP : ARRAY  [1 .. 40 ] OF BYTE ;
   END_STRUCT ;
  END_STRUCT ;
BEGIN
   S700_BT_CODE_2011.STATION_MAIN := W#16#0;
   S700_BT_CODE_2011.DISTINCTION_LH_RH := W#16#0;
   S700_BT_CODE_2011.STAION_NUMBER := W#16#0;
   S700_BT_CODE_2011.BODY_TYPE_1ST := W#16#0;
   S700_BT_CODE_2011.BODY_TYPE_OPTION := W#16#0;
   S700_BT_CODE_2011.RBT1_STANDARD_WELD_DATA := W#16#0;
   S700_BT_CODE_2011.RBT2_STANDARD_WELD_DATA := W#16#0;
   S700_BT_CODE_2011.RBT3_STANDARD_WELD_DATA := W#16#0;
   S700_BT_CODE_2011.RBT4_STANDARD_WELD_DATA := W#16#0;
   S700_BT_CODE_2011.RBT5_STANDARD_WELD_DATA := W#16#0;
   S700_BT_CODE_2011.RBT6_STANDARD_WELD_DATA := W#16#0;
   S700_BT_CODE_2011.RBT7_STANDARD_WELD_DATA := W#16#0;
   S700_BT_CODE_2011.RBT8_STANDARD_WELD_DATA := W#16#0;
   S700_BT_CODE_2011.RBT9_STANDARD_WELD_DATA := W#16#0;
   S700_BT_CODE_2011.RBT10_STANDARD_WELD_DATA := W#16#0;
   S700_BT_CODE_2011.RBT11_STANDARD_WELD_DATA := W#16#0;
   S700_BT_CODE_2011.RBT12_STANDARD_WELD_DATA := W#16#0;
   S700_BT_CODE_2011.RBT13_STANDARD_WELD_DATA := W#16#0;
   S700_BT_CODE_2011.RBT14_STANDARD_WELD_DATA := W#16#0;
   S700_BT_CODE_2011.RBT15_STANDARD_WELD_DATA := W#16#0;
   S700_BT_CODE_2011.RBT16_STANDARD_WELD_DATA := W#16#0;
   S700_BT_CODE_2011.RBT17_STANDARD_WELD_DATA := W#16#0;
   S700_BT_CODE_2011.RBT18_STANDARD_WELD_DATA := W#16#0;
   S700_BT_CODE_2011.RBT19_STANDARD_WELD_DATA := W#16#0;
   S700_BT_CODE_2011.RBT20_STANDARD_WELD_DATA := W#16#0;
   S700_BT_CODE_2011.RBT21_STANDARD_WELD_DATA := W#16#0;
   S700_BT_CODE_2011.RBT22_STANDARD_WELD_DATA := W#16#0;
   S700_BT_CODE_2011.RBT23_STANDARD_WELD_DAT := W#16#0;
   S700_BT_CODE_2011.RBT24_STANDARD_WELD_DAT := W#16#0;
   S700_BT_CODE_2011.CHK_WORD := W#16#0;
   S700_BT_CODE_2011.TEST_TEMP[1] := B#16#0;
   S700_BT_CODE_2011.TEST_TEMP[2] := B#16#0;
   S700_BT_CODE_2011.TEST_TEMP[3] := B#16#0;
   S700_BT_CODE_2011.TEST_TEMP[4] := B#16#0;
   S700_BT_CODE_2011.TEST_TEMP[5] := B#16#0;
   S700_BT_CODE_2011.TEST_TEMP[6] := B#16#0;
   S700_BT_CODE_2011.TEST_TEMP[7] := B#16#0;
   S700_BT_CODE_2011.TEST_TEMP[8] := B#16#0;
   S700_BT_CODE_2011.TEST_TEMP[9] := B#16#0;
   S700_BT_CODE_2011.TEST_TEMP[10] := B#16#0;
   S700_BT_CODE_2011.TEST_TEMP[11] := B#16#0;
   S700_BT_CODE_2011.TEST_TEMP[12] := B#16#0;
   S700_BT_CODE_2011.TEST_TEMP[13] := B#16#0;
   S700_BT_CODE_2011.TEST_TEMP[14] := B#16#0;
   S700_BT_CODE_2011.TEST_TEMP[15] := B#16#0;
   S700_BT_CODE_2011.TEST_TEMP[16] := B#16#0;
   S700_BT_CODE_2011.TEST_TEMP[17] := B#16#0;
   S700_BT_CODE_2011.TEST_TEMP[18] := B#16#0;
   S700_BT_CODE_2011.TEST_TEMP[19] := B#16#0;
   S700_BT_CODE_2011.TEST_TEMP[20] := B#16#0;
   S700_BT_CODE_2011.TEST_TEMP[21] := B#16#0;
   S700_BT_CODE_2011.TEST_TEMP[22] := B#16#0;
   S700_BT_CODE_2011.TEST_TEMP[23] := B#16#0;
   S700_BT_CODE_2011.TEST_TEMP[24] := B#16#0;
   S700_BT_CODE_2011.TEST_TEMP[25] := B#16#0;
   S700_BT_CODE_2011.TEST_TEMP[26] := B#16#0;
   S700_BT_CODE_2011.TEST_TEMP[27] := B#16#0;
   S700_BT_CODE_2011.TEST_TEMP[28] := B#16#0;
   S700_BT_CODE_2011.TEST_TEMP[29] := B#16#0;
   S700_BT_CODE_2011.TEST_TEMP[30] := B#16#0;
   S700_BT_CODE_2011.TEST_TEMP[31] := B#16#0;
   S700_BT_CODE_2011.TEST_TEMP[32] := B#16#0;
   S700_BT_CODE_2011.TEST_TEMP[33] := B#16#0;
   S700_BT_CODE_2011.TEST_TEMP[34] := B#16#0;
   S700_BT_CODE_2011.TEST_TEMP[35] := B#16#0;
   S700_BT_CODE_2011.TEST_TEMP[36] := B#16#0;
   S700_BT_CODE_2011.TEST_TEMP[37] := B#16#0;
   S700_BT_CODE_2011.TEST_TEMP[38] := B#16#0;
   S700_BT_CODE_2011.TEST_TEMP[39] := B#16#0;
   S700_BT_CODE_2011.TEST_TEMP[40] := B#16#0;
   S700_BT_CODE_2012.STATION_MAIN := W#16#0;
   S700_BT_CODE_2012.DISTINCTION_LH_RH := W#16#0;
   S700_BT_CODE_2012.STAION_NUMBER := W#16#0;
   S700_BT_CODE_2012.BODY_TYPE_1ST := W#16#0;
   S700_BT_CODE_2012.BODY_TYPE_OPTION := W#16#0;
   S700_BT_CODE_2012.RBT1_STANDARD_WELD_DATA := W#16#0;
   S700_BT_CODE_2012.RBT2_STANDARD_WELD_DATA := W#16#0;
   S700_BT_CODE_2012.RBT3_STANDARD_WELD_DATA := W#16#0;
   S700_BT_CODE_2012.RBT4_STANDARD_WELD_DATA := W#16#0;
   S700_BT_CODE_2012.RBT5_STANDARD_WELD_DATA := W#16#0;
   S700_BT_CODE_2012.RBT6_STANDARD_WELD_DATA := W#16#0;
   S700_BT_CODE_2012.RBT7_STANDARD_WELD_DATA := W#16#0;
   S700_BT_CODE_2012.RBT8_STANDARD_WELD_DATA := W#16#0;
   S700_BT_CODE_2012.RBT9_STANDARD_WELD_DATA := W#16#0;
   S700_BT_CODE_2012.RBT10_STANDARD_WELD_DATA := W#16#0;
   S700_BT_CODE_2012.RBT11_STANDARD_WELD_DATA := W#16#0;
   S700_BT_CODE_2012.RBT12_STANDARD_WELD_DATA := W#16#0;
   S700_BT_CODE_2012.RBT13_STANDARD_WELD_DATA := W#16#0;
   S700_BT_CODE_2012.RBT14_STANDARD_WELD_DATA := W#16#0;
   S700_BT_CODE_2012.RBT15_STANDARD_WELD_DATA := W#16#0;
   S700_BT_CODE_2012.RBT16_STANDARD_WELD_DATA := W#16#0;
   S700_BT_CODE_2012.RBT17_STANDARD_WELD_DATA := W#16#0;
   S700_BT_CODE_2012.RBT18_STANDARD_WELD_DATA := W#16#0;
   S700_BT_CODE_2012.RBT19_STANDARD_WELD_DATA := W#16#0;
   S700_BT_CODE_2012.RBT20_STANDARD_WELD_DATA := W#16#0;
   S700_BT_CODE_2012.RBT21_STANDARD_WELD_DATA := W#16#0;
   S700_BT_CODE_2012.RBT22_STANDARD_WELD_DATA := W#16#0;
   S700_BT_CODE_2012.RBT23_STANDARD_WELD_DAT := W#16#0;
   S700_BT_CODE_2012.RBT24_STANDARD_WELD_DAT := W#16#0;
   S700_BT_CODE_2012.CHK_WORD := W#16#0;
   S700_BT_CODE_2012.TEST_TEMP[1] := B#16#0;
   S700_BT_CODE_2012.TEST_TEMP[2] := B#16#0;
   S700_BT_CODE_2012.TEST_TEMP[3] := B#16#0;
   S700_BT_CODE_2012.TEST_TEMP[4] := B#16#0;
   S700_BT_CODE_2012.TEST_TEMP[5] := B#16#0;
   S700_BT_CODE_2012.TEST_TEMP[6] := B#16#0;
   S700_BT_CODE_2012.TEST_TEMP[7] := B#16#0;
   S700_BT_CODE_2012.TEST_TEMP[8] := B#16#0;
   S700_BT_CODE_2012.TEST_TEMP[9] := B#16#0;
   S700_BT_CODE_2012.TEST_TEMP[10] := B#16#0;
   S700_BT_CODE_2012.TEST_TEMP[11] := B#16#0;
   S700_BT_CODE_2012.TEST_TEMP[12] := B#16#0;
   S700_BT_CODE_2012.TEST_TEMP[13] := B#16#0;
   S700_BT_CODE_2012.TEST_TEMP[14] := B#16#0;
   S700_BT_CODE_2012.TEST_TEMP[15] := B#16#0;
   S700_BT_CODE_2012.TEST_TEMP[16] := B#16#0;
   S700_BT_CODE_2012.TEST_TEMP[17] := B#16#0;
   S700_BT_CODE_2012.TEST_TEMP[18] := B#16#0;
   S700_BT_CODE_2012.TEST_TEMP[19] := B#16#0;
   S700_BT_CODE_2012.TEST_TEMP[20] := B#16#0;
   S700_BT_CODE_2012.TEST_TEMP[21] := B#16#0;
   S700_BT_CODE_2012.TEST_TEMP[22] := B#16#0;
   S700_BT_CODE_2012.TEST_TEMP[23] := B#16#0;
   S700_BT_CODE_2012.TEST_TEMP[24] := B#16#0;
   S700_BT_CODE_2012.TEST_TEMP[25] := B#16#0;
   S700_BT_CODE_2012.TEST_TEMP[26] := B#16#0;
   S700_BT_CODE_2012.TEST_TEMP[27] := B#16#0;
   S700_BT_CODE_2012.TEST_TEMP[28] := B#16#0;
   S700_BT_CODE_2012.TEST_TEMP[29] := B#16#0;
   S700_BT_CODE_2012.TEST_TEMP[30] := B#16#0;
   S700_BT_CODE_2012.TEST_TEMP[31] := B#16#0;
   S700_BT_CODE_2012.TEST_TEMP[32] := B#16#0;
   S700_BT_CODE_2012.TEST_TEMP[33] := B#16#0;
   S700_BT_CODE_2012.TEST_TEMP[34] := B#16#0;
   S700_BT_CODE_2012.TEST_TEMP[35] := B#16#0;
   S700_BT_CODE_2012.TEST_TEMP[36] := B#16#0;
   S700_BT_CODE_2012.TEST_TEMP[37] := B#16#0;
   S700_BT_CODE_2012.TEST_TEMP[38] := B#16#0;
   S700_BT_CODE_2012.TEST_TEMP[39] := B#16#0;
   S700_BT_CODE_2012.TEST_TEMP[40] := B#16#0;
   S700_BT_CODE_2013.STATION_MAIN := W#16#0;
   S700_BT_CODE_2013.DISTINCTION_LH_RH := W#16#0;
   S700_BT_CODE_2013.STAION_NUMBER := W#16#0;
   S700_BT_CODE_2013.BODY_TYPE_1ST := W#16#0;
   S700_BT_CODE_2013.BODY_TYPE_OPTION := W#16#0;
   S700_BT_CODE_2013.RBT1_STANDARD_WELD_DATA := W#16#0;
   S700_BT_CODE_2013.RBT2_STANDARD_WELD_DATA := W#16#0;
   S700_BT_CODE_2013.RBT3_STANDARD_WELD_DATA := W#16#0;
   S700_BT_CODE_2013.RBT4_STANDARD_WELD_DATA := W#16#0;
   S700_BT_CODE_2013.RBT5_STANDARD_WELD_DATA := W#16#0;
   S700_BT_CODE_2013.RBT6_STANDARD_WELD_DATA := W#16#0;
   S700_BT_CODE_2013.RBT7_STANDARD_WELD_DATA := W#16#0;
   S700_BT_CODE_2013.RBT8_STANDARD_WELD_DATA := W#16#0;
   S700_BT_CODE_2013.RBT9_STANDARD_WELD_DATA := W#16#0;
   S700_BT_CODE_2013.RBT10_STANDARD_WELD_DATA := W#16#0;
   S700_BT_CODE_2013.RBT11_STANDARD_WELD_DATA := W#16#0;
   S700_BT_CODE_2013.RBT12_STANDARD_WELD_DATA := W#16#0;
   S700_BT_CODE_2013.RBT13_STANDARD_WELD_DATA := W#16#0;
   S700_BT_CODE_2013.RBT14_STANDARD_WELD_DATA := W#16#0;
   S700_BT_CODE_2013.RBT15_STANDARD_WELD_DATA := W#16#0;
   S700_BT_CODE_2013.RBT16_STANDARD_WELD_DATA := W#16#0;
   S700_BT_CODE_2013.RBT17_STANDARD_WELD_DATA := W#16#0;
   S700_BT_CODE_2013.RBT18_STANDARD_WELD_DATA := W#16#0;
   S700_BT_CODE_2013.RBT19_STANDARD_WELD_DATA := W#16#0;
   S700_BT_CODE_2013.RBT20_STANDARD_WELD_DATA := W#16#0;
   S700_BT_CODE_2013.RBT21_STANDARD_WELD_DATA := W#16#0;
   S700_BT_CODE_2013.RBT22_STANDARD_WELD_DATA := W#16#0;
   S700_BT_CODE_2013.RBT23_STANDARD_WELD_DAT := W#16#0;
   S700_BT_CODE_2013.RBT24_STANDARD_WELD_DAT := W#16#0;
   S700_BT_CODE_2013.CHK_WORD := W#16#0;
   S700_BT_CODE_2013.TEST_TEMP[1] := B#16#0;
   S700_BT_CODE_2013.TEST_TEMP[2] := B#16#0;
   S700_BT_CODE_2013.TEST_TEMP[3] := B#16#0;
   S700_BT_CODE_2013.TEST_TEMP[4] := B#16#0;
   S700_BT_CODE_2013.TEST_TEMP[5] := B#16#0;
   S700_BT_CODE_2013.TEST_TEMP[6] := B#16#0;
   S700_BT_CODE_2013.TEST_TEMP[7] := B#16#0;
   S700_BT_CODE_2013.TEST_TEMP[8] := B#16#0;
   S700_BT_CODE_2013.TEST_TEMP[9] := B#16#0;
   S700_BT_CODE_2013.TEST_TEMP[10] := B#16#0;
   S700_BT_CODE_2013.TEST_TEMP[11] := B#16#0;
   S700_BT_CODE_2013.TEST_TEMP[12] := B#16#0;
   S700_BT_CODE_2013.TEST_TEMP[13] := B#16#0;
   S700_BT_CODE_2013.TEST_TEMP[14] := B#16#0;
   S700_BT_CODE_2013.TEST_TEMP[15] := B#16#0;
   S700_BT_CODE_2013.TEST_TEMP[16] := B#16#0;
   S700_BT_CODE_2013.TEST_TEMP[17] := B#16#0;
   S700_BT_CODE_2013.TEST_TEMP[18] := B#16#0;
   S700_BT_CODE_2013.TEST_TEMP[19] := B#16#0;
   S700_BT_CODE_2013.TEST_TEMP[20] := B#16#0;
   S700_BT_CODE_2013.TEST_TEMP[21] := B#16#0;
   S700_BT_CODE_2013.TEST_TEMP[22] := B#16#0;
   S700_BT_CODE_2013.TEST_TEMP[23] := B#16#0;
   S700_BT_CODE_2013.TEST_TEMP[24] := B#16#0;
   S700_BT_CODE_2013.TEST_TEMP[25] := B#16#0;
   S700_BT_CODE_2013.TEST_TEMP[26] := B#16#0;
   S700_BT_CODE_2013.TEST_TEMP[27] := B#16#0;
   S700_BT_CODE_2013.TEST_TEMP[28] := B#16#0;
   S700_BT_CODE_2013.TEST_TEMP[29] := B#16#0;
   S700_BT_CODE_2013.TEST_TEMP[30] := B#16#0;
   S700_BT_CODE_2013.TEST_TEMP[31] := B#16#0;
   S700_BT_CODE_2013.TEST_TEMP[32] := B#16#0;
   S700_BT_CODE_2013.TEST_TEMP[33] := B#16#0;
   S700_BT_CODE_2013.TEST_TEMP[34] := B#16#0;
   S700_BT_CODE_2013.TEST_TEMP[35] := B#16#0;
   S700_BT_CODE_2013.TEST_TEMP[36] := B#16#0;
   S700_BT_CODE_2013.TEST_TEMP[37] := B#16#0;
   S700_BT_CODE_2013.TEST_TEMP[38] := B#16#0;
   S700_BT_CODE_2013.TEST_TEMP[39] := B#16#0;
   S700_BT_CODE_2013.TEST_TEMP[40] := B#16#0;
   S700_BT_CODE_2014.STATION_MAIN := W#16#0;
   S700_BT_CODE_2014.DISTINCTION_LH_RH := W#16#0;
   S700_BT_CODE_2014.STAION_NUMBER := W#16#0;
   S700_BT_CODE_2014.BODY_TYPE_1ST := W#16#0;
   S700_BT_CODE_2014.BODY_TYPE_OPTION := W#16#0;
   S700_BT_CODE_2014.RBT1_STANDARD_WELD_DATA := W#16#0;
   S700_BT_CODE_2014.RBT2_STANDARD_WELD_DATA := W#16#0;
   S700_BT_CODE_2014.RBT3_STANDARD_WELD_DATA := W#16#0;
   S700_BT_CODE_2014.RBT4_STANDARD_WELD_DATA := W#16#0;
   S700_BT_CODE_2014.RBT5_STANDARD_WELD_DATA := W#16#0;
   S700_BT_CODE_2014.RBT6_STANDARD_WELD_DATA := W#16#0;
   S700_BT_CODE_2014.RBT7_STANDARD_WELD_DATA := W#16#0;
   S700_BT_CODE_2014.RBT8_STANDARD_WELD_DATA := W#16#0;
   S700_BT_CODE_2014.RBT9_STANDARD_WELD_DATA := W#16#0;
   S700_BT_CODE_2014.RBT10_STANDARD_WELD_DATA := W#16#0;
   S700_BT_CODE_2014.RBT11_STANDARD_WELD_DATA := W#16#0;
   S700_BT_CODE_2014.RBT12_STANDARD_WELD_DATA := W#16#0;
   S700_BT_CODE_2014.RBT13_STANDARD_WELD_DATA := W#16#0;
   S700_BT_CODE_2014.RBT14_STANDARD_WELD_DATA := W#16#0;
   S700_BT_CODE_2014.RBT15_STANDARD_WELD_DATA := W#16#0;
   S700_BT_CODE_2014.RBT16_STANDARD_WELD_DATA := W#16#0;
   S700_BT_CODE_2014.RBT17_STANDARD_WELD_DATA := W#16#0;
   S700_BT_CODE_2014.RBT18_STANDARD_WELD_DATA := W#16#0;
   S700_BT_CODE_2014.RBT19_STANDARD_WELD_DATA := W#16#0;
   S700_BT_CODE_2014.RBT20_STANDARD_WELD_DATA := W#16#0;
   S700_BT_CODE_2014.RBT21_STANDARD_WELD_DATA := W#16#0;
   S700_BT_CODE_2014.RBT22_STANDARD_WELD_DATA := W#16#0;
   S700_BT_CODE_2014.RBT23_STANDARD_WELD_DAT := W#16#0;
   S700_BT_CODE_2014.RBT24_STANDARD_WELD_DAT := W#16#0;
   S700_BT_CODE_2014.CHK_WORD := W#16#0;
   S700_BT_CODE_2014.TEST_TEMP[1] := B#16#0;
   S700_BT_CODE_2014.TEST_TEMP[2] := B#16#0;
   S700_BT_CODE_2014.TEST_TEMP[3] := B#16#0;
   S700_BT_CODE_2014.TEST_TEMP[4] := B#16#0;
   S700_BT_CODE_2014.TEST_TEMP[5] := B#16#0;
   S700_BT_CODE_2014.TEST_TEMP[6] := B#16#0;
   S700_BT_CODE_2014.TEST_TEMP[7] := B#16#0;
   S700_BT_CODE_2014.TEST_TEMP[8] := B#16#0;
   S700_BT_CODE_2014.TEST_TEMP[9] := B#16#0;
   S700_BT_CODE_2014.TEST_TEMP[10] := B#16#0;
